(* CODESYS project CtaAppStufenManagement_4.0.0.1.library
   Description: Stufenmanagement Library der CTA
   Version: 4.0.0.1
   Title: CtaAppStufenManagement
   Author: SIS
   DocFormat: reStructuredText
   LanguageModelAttribute: qualified-access-only
   Placeholder: CtaAppStufenManagement
   DefaultNamespace: CtaAppStufenManagement
   CompiledLibraryCompatibilityVersion: CODESYS V3.5 SP16 Patch 3
   Company: CTA

Project tree, tasks and I/O mapping:
  libraries: Standard, 3.5.18.0 (System); CtaAppBasic, 1.0.0.1 (CTA); CtaAppBmk, 2.0.0.0 (CTA); CtaSysConfig, 2.0.0.0 (CTA); VisuDialogs, 3.5.16.20 (System); VisuSymbols, 4.5.0.0 (System); CtaVisHelp, 2.0.0.0 (CTA); CtaVisSymbols, 2.0.0.1 (CTA); CtaSysTypes, 1.0.0.0 (CTA)
  40 Visualizations/
    visualisation VIS_Manager_rEck
    Dialog/
      visualisation DIA_MANAGERCONFIG
    visualisation VIS_Manager
  00000000-0000-0000-0000-000000000000|D:\CoDeSys\LibrariesV3\trunk\Intern\CAA\CAA Template\3.4.0.0 draft\Placeholder.xml
  00000000-0000-0000-0000-000000000000|D:\CoDeSys\LibrariesV3\trunk\Intern\CAA\CAA Template\3.2.0.3 draft\Prefix.pdf
  00000000-0000-0000-0000-000000000000|D:\CoDeSys\LibrariesV3\trunk\Intern\CAA\CAA Template\3.5.2.0 draft\Placeholder.xml
  20 Structs/
    data type TYPE_OF_ENGINE_MANAGEMENT
    data type scParameter
  50 Images/
  10 Documenation/
    global variables VersionHistory
    global variables readMe
  21 Interface/
    Group/
      GroupBase/
        interface ITF_GROUPBASE: IS_NOT_RELEVANT_TO_CHECK, set_acknowledge_substate, acknowledge_substate, acknowledge, set_acknowledge, acknowledge_old, acknowledge_substate_old, IS_NOT_RELEVANT_TO_RELEASE, IS_ADDED_TO_NESSESARY, check, set_check, set_check_substate, check_substate, check_old, check_substate_old, release, set_release, set_release_next, set_release_substate, release_substate, release_old, release_substate_old, release_next, release_next_old, IS_NOT_RELEVANT_TO_ACKNOWLEDGE, available_substate, set_available_substate, set_available, available, available_old, available_substate_old, set_demand, demand, demand_old
      GroupLeader/
        Circuit/
          interface ITF_CIRCUIT: GET_ANZ_AVAIABLE, GET_ANZ_ACKNOWLEDGE, GET_ANZ_RELEASE, CIRCUIT_NR, ALL_OFF, IS_RELEVANT_TO_RELEASE, GET_ENGINE_STATE, RELEASE_ENGINE, LOWERBOUND, UPPERBOUND, GET_ANZ_LOCKDOWN, SET_HZ_SCALE, SET_ENGINE_STATE, prorRelease, GET_SUM_ACKNOWLEDGE_HZ
      GroupMember/
        Hydraulics/
          interface ITF_HYDRA: MEMBER_OF
    Manager/
      interface ITF_MANAGER: ADD_CLIENT
  11 Library Parameter/
  12 Konstanten/
    global variables GVL_CONSTANT
  60 Textlisten/
    text list TypeOfEngineManagement
  13 Globale Variablen/
  text list GlobalTextList
  5ce3da45-db07-42e7-a21c-a00fff4ed8f6|C:\Users\sis\Downloads\dip-switch.svg
  5ce3da45-db07-42e7-a21c-a00fff4ed8f6|C:\Users\sis\Downloads\lightning-bolt-circle.svg
  30 Program Organization Units/
    Group/
      GroupBase/
        function block GROUPBASE [ST]: IS_NOT_RELEVANT_TO_CHECK, IS_NOT_RELEVANT_TO_RELEASE, set_acknowledge, set_acknowledge_substate, acknowledge, acknowledge_substate, acknowledge_old, acknowledge_substate_old, available_substate, available, set_available, set_available_substate, available_old, available_substate_old, check_substate, set_check_substate, check, set_check, check_old, check_substate_old, set_release_next, release, release_substate, set_release, set_release_substate, release_next, release_next_old, release_old, release_substate_old, IS_NOT_RELEVANT_TO_ACKNOWLEDGE, set_demand, demand, demand_old, IS_ADDED_TO_NESSESARY
      GroupLeader/
        Help/
          function block ENGINE [ST]: GET_ANZ_AVAIABLE, GET_ANZ_ACKNOWLEDGE, GET_ANZ_RELEASE, GET_ANZ_LOCKDOWN, SET_ENGINE_STATE, GET_ENGINE_STATE, RELEASE_ENGINE, LOWERBOUND, UPPERBOUND, SET_HZ_SCALE, GET_ANZ_ENABLED, GET_SUM_ACKNOWLEDGE_HZ
        Circuit/
          function block CIRCUIT [ST]: IS_RELEVANT_TO_RELEASE, SET_ENGINE_STATE, GET_ANZ_AVAIABLE, GET_ANZ_ACKNOWLEDGE, GET_ANZ_RELEASE, CIRCUIT_NR, ALL_OFF, GET_ENGINE_STATE, RELEASE_ENGINE, LOWERBOUND, UPPERBOUND, GET_ANZ_LOCKDOWN, SET_HZ_SCALE, prorRelease, GET_ANZ_ENABLED, GET_SUM_ACKNOWLEDGE_HZ
      GroupMember/
        Help/
          function block GROUPMEMBER [ST]
        Hydraulics/
          function block HYDRA [ST]: MEMBER_OF, FB_INIT
    Manager/
      function block MANAGER [ST]: CHECK, set_check_of_group, set_check_substate_of_group, get_next_engine_to_start, get_next_engine_to_stopp, engine_management_start_run_1_by_1, engine_management_start_run_equal, engine_management_stopp_run_1_by_1, engine_management_stopp_run_equal, ENGINE_MANAGEMENT, UPDATE_AT_THE_END, ACKNOWLEDGE, check_acknowledge_of_group, check_acknowledge_substate_of_group, RELEASE, set_release_of_group, set_release_substate_of_group, set_release_next_of_group, LOCKDOWN, AVAIABLE, check_available_of_group, check_available_substate_of_group, ADD_CLIENT, actParameter, FB_INIT, DEMAND, set_priority_array, init_priority_array_with_ignore_state
  5ce3da45-db07-42e7-a21c-a00fff4ed8f6|C:\Users\sis\Downloads\sine-wave.svg
  5ce3da45-db07-42e7-a21c-a00fff4ed8f6|C:\Users\sis\Downloads\eye.svg
  5ce3da45-db07-42e7-a21c-a00fff4ed8f6|C:\Users\sis\Downloads\lan.svg
*)

// 20 Structs/TYPE_OF_ENGINE_MANAGEMENT
{attribute 'qualified_only'}
TYPE TYPE_OF_ENGINE_MANAGEMENT :
(
	RUN_1BY1 	:= 0,
	RUN_EQUAL	:= 1
);
END_TYPE

// 20 Structs/scParameter
TYPE scParameter :
	STRUCT
		fbtZuschaltSperrzeit		:	CtaSysConfig.fbTIME;
		fbiTypeOfEngineManagement	:	CtaSysConfig.fbINT;
	END_STRUCT
END_TYPE

// 10 Documenation/VersionHistory
(* 

.. image:: ../../Images/CTA_Logo.jpg
   :align: right
   :width: 15% 

**Vorlage**   


============ =========== =========== ============================================
**Date**     **Version** **Author**  **Change**
------------ ----------- ----------- --------------------------------------------
04.03.2021   0.0.0.0     SIS         Vorlage erstellt

============ =========== =========== ============================================


*)
VAR_GLOBAL
    stInfo : STRING:= '0.0.0.0, Vorlage, CTA';
END_VAR

// 10 Documenation/readMe
(*

**ReadMe**
 
|	**Empfehlung**
|
|	Die Bibliothek CtaAppStufenManagement dient dem Management der ganzen Maschine, sie Schaltet beispielsweise Kreise und Stufen frei.
|	Instanzieren Sie den CtaAppStufenManagement.MANAGER in ihrem Funktionsbaustein oder POU beispielsweise als Manager
|	Deklarieren Sie die Struktur Variable welche als Parameter und zur ansteuerung dienen wie im Code beispiel.
|  
| *Beispiel* 

+-----------------------+---------------------------------------------------------------------------------------------------------------------------------------------------------------------------------------------------------------------------------------------------------------------------------------------------------------------------------------------------------------------------------------------------------------------------------------+
| Beschreibung          |  Code                                                                                                                                                                                                                                                                                                                                                                                                                                 |
+=======================+=======================================================================================================================================================================================================================================================================================================================================================================================================================================+
| Pou oder SmFb         | .. code-block:: codesys                                                                                                                                                                                                                                                                                                                                                                                                               |
|                       |                                                                                                                                                                                                                                                                                                                                                                                                                                       |
|                       |	// Deklaration als VAR im POU oder dem selbsterstellten Funktionsbaustein                                                                                                                                                                                                                                                                                                                                                       	|
|                       |   VAR   																																																																																																								|
|						|	    (*Maschinen Management*)																																																		 																																																|
|						|		MANAGER			: CtaAppStufenManagement.MANAGER;                                                                                                                                                                                                                                                                                                                                                             				 	|
|						|																																																																																																										|
+-----------------------+---------------------------------------------------------------------------------------------------------------------------------------------------------------------------------------------------------------------------------------------------------------------------------------------------------------------------------------------------------------------------------------------------------------------------------------+
| Code für Init         | .. code-block:: codesys                                                                                                                                                                                                                                                                                                                                                                                                               |
|                       |   																																																																																																									|
| 						|	// Kopieren des nachfolgenden Codes in eine Action zur Initialisierung der Parameter. Zum Beispiel actConfig.																																																																														|
|                       |	{region "Maschinen Management"}                                                                                                                                                                                                                                                                                                                                                                                                     |
|						|		MANAGER.scParameter.fbtZuschaltSperrzeit               		(_wertInit :=	 T#5m														);		//P1 Zeit die vergeht bis die nächste Stufe zugeschalten werden kann																																																			|
|						|		MANAGER.scParameter.fbiTypeOfEngineManagement				(_wertInit :=	 	0		, _minInit :=			, _maxInit :=			);		//P2 0 = Ausschöpfung des Kreises / 1 = Beliebig nach verfügbarkeit																																																				| 
|						|	{endregion}                                                                                                                                                      																																																																	| 
+-----------------------+---------------------------------------------------------------------------------------------------------------------------------------------------------------------------------------------------------------------------------------------------------------------------------------------------------------------------------------------------------------------------------------------------------------------------------------+
*)                                                                                                                                                                                                                                                                                                                                                                                                                                                               
 VAR_GLOBAL                                                                                                                                                                                                                                                                                                                                                                                                                                                      
    xReadMeDone              :   BOOL;                                                                                                                                                                                                                                                                                                                                                                                                                           
END_VAR

// 12 Konstanten/GVL_CONSTANT
{attribute 'qualified_only'}
VAR_GLOBAL CONSTANT
	MAX_GROUPS	:	USINT	:= 4;
	MAX_ENGINE	:	USINT	:= 4;
END_VAR

// 21 Interface/Group/GroupBase/ITF_GROUPBASE
INTERFACE ITF_GROUPBASE EXTENDS __SYSTEM.IQueryInterface

{attribute 'monitoring':='call'}
PROPERTY IS_NOT_RELEVANT_TO_CHECK : BOOL
GET
END_GET
SET
END_SET
END_PROPERTY

METHOD set_acknowledge_substate
VAR_INPUT
	_en_acknowledge_substate		:	INT;
END_VAR
END_METHOD

{attribute 'monitoring':='call'}
PROPERTY acknowledge_substate : INT
GET
END_GET
END_PROPERTY

{attribute 'monitoring':='call'}
PROPERTY acknowledge : INT
GET
END_GET
END_PROPERTY

METHOD set_acknowledge
VAR_INPUT
	_en_acknowledge		:	INT;
END_VAR
END_METHOD

{attribute 'monitoring':='call'}
PROPERTY acknowledge_old : INT
GET
END_GET
END_PROPERTY

{attribute 'monitoring':='call'}
PROPERTY acknowledge_substate_old : INT
GET
END_GET
END_PROPERTY

{attribute 'monitoring':='call'}
PROPERTY IS_NOT_RELEVANT_TO_RELEASE : BOOL
GET
END_GET
SET
END_SET
END_PROPERTY

PROPERTY IS_ADDED_TO_NESSESARY : BOOL
SET
END_SET
GET
END_GET
END_PROPERTY

{attribute 'monitoring':='call'}
PROPERTY check : INT
GET
END_GET
END_PROPERTY

METHOD set_check
VAR_INPUT
	_en_check			:	INT;
END_VAR
END_METHOD

METHOD set_check_substate
VAR_INPUT
	_en_check_substate				:	INT;
END_VAR
END_METHOD

{attribute 'monitoring':='call'}
PROPERTY check_substate : INT
GET
END_GET
END_PROPERTY

{attribute 'monitoring':='call'}
PROPERTY check_old : INT
GET
END_GET
END_PROPERTY

{attribute 'monitoring':='call'}
PROPERTY check_substate_old : INT
GET
END_GET
END_PROPERTY

{attribute 'monitoring':='call'}
PROPERTY release : INT
GET
END_GET
END_PROPERTY

METHOD set_release
VAR_INPUT
	_en_release			:	INT;
END_VAR
END_METHOD

METHOD set_release_next
VAR_INPUT
	_en_release_next	:	INT;
END_VAR
END_METHOD

METHOD set_release_substate
VAR_INPUT
	_en_release_substate	:	INT;
END_VAR
END_METHOD

{attribute 'monitoring':='call'}
PROPERTY release_substate : INT
GET
END_GET
END_PROPERTY

{attribute 'monitoring':='call'}
PROPERTY release_old : INT
GET
END_GET
END_PROPERTY

{attribute 'monitoring':='call'}
PROPERTY release_substate_old : INT
GET
END_GET
END_PROPERTY

PROPERTY release_next : INT
GET
END_GET
END_PROPERTY

PROPERTY release_next_old : INT
GET
END_GET
END_PROPERTY

{attribute 'monitoring':='call'}
PROPERTY IS_NOT_RELEVANT_TO_ACKNOWLEDGE : BOOL
SET
END_SET
GET
END_GET
END_PROPERTY

{attribute 'monitoring':='call'}
PROPERTY available_substate : INT
GET
END_GET
END_PROPERTY

METHOD set_available_substate
VAR_INPUT
	_en_avaiable_substate	:	INT;
END_VAR
END_METHOD

METHOD set_available
VAR_INPUT
	_en_avaiable		:	INT;
END_VAR
END_METHOD

{attribute 'monitoring':='call'}
PROPERTY available : INT
GET
END_GET
END_PROPERTY

{attribute 'monitoring':='call'}
PROPERTY available_old : INT
GET
END_GET
END_PROPERTY

{attribute 'monitoring':='call'}
PROPERTY available_substate_old : INT
GET
END_GET
END_PROPERTY

METHOD set_demand
VAR_INPUT
	_en_demand			:	INT;
END_VAR
END_METHOD

{attribute 'monitoring':='call'}
PROPERTY demand : INT
GET
END_GET
END_PROPERTY

{attribute 'monitoring':='call'}
PROPERTY demand_old : INT
GET
END_GET
END_PROPERTY

END_INTERFACE

// 21 Interface/Manager/ITF_MANAGER
INTERFACE ITF_MANAGER EXTENDS __SYSTEM.IQueryInterface

METHOD ADD_CLIENT : BOOL
VAR_INPUT
	ITF_GROUP_BASE_IN	:	ITF_GROUPBASE;
END_VAR
END_METHOD

END_INTERFACE

// 21 Interface/Group/GroupLeader/Circuit/ITF_CIRCUIT
INTERFACE ITF_CIRCUIT EXTENDS ITF_GROUPBASE

PROPERTY GET_ANZ_AVAIABLE : UINT
GET
END_GET
END_PROPERTY

PROPERTY GET_ANZ_ACKNOWLEDGE : UINT
GET
END_GET
END_PROPERTY

PROPERTY GET_ANZ_RELEASE : UINT
GET
END_GET
END_PROPERTY

PROPERTY CIRCUIT_NR : USINT
GET
END_GET
END_PROPERTY

METHOD ALL_OFF : BOOL
VAR_INPUT
END_VAR
END_METHOD

PROPERTY IS_RELEVANT_TO_RELEASE : BOOL
GET
END_GET
SET
END_SET
END_PROPERTY

METHOD GET_ENGINE_STATE : BOOL
VAR_INPUT
	usiNr				:	USINT;
END_VAR
VAR_OUTPUT	    	
	xAvaiable			:	BOOL;
	xRelease			:	BOOL;
	rRelease			:	REAL;
	xAcknowledge		:	BOOL;
	rAcknowledgeHz		:	REAL;
	xLockDown			:	BOOL;
	udiRunTime			:	UDINT;
	udiRunTimeTillOn	:	UDINT;
END_VAR
END_METHOD

METHOD RELEASE_ENGINE
VAR_INPUT
	usiNr		:	USINT;
	xRelease	:	BOOL;
END_VAR
END_METHOD

PROPERTY LOWERBOUND : DINT
GET
END_GET
END_PROPERTY

PROPERTY UPPERBOUND : DINT
GET
END_GET
END_PROPERTY

PROPERTY GET_ANZ_LOCKDOWN : UINT
GET
END_GET
END_PROPERTY

METHOD SET_HZ_SCALE
VAR_INPUT
	scHz		:	CtaSysTypes.scHzParameter;
END_VAR
END_METHOD

METHOD SET_ENGINE_STATE 
VAR_INPUT
	usiNr		:	USINT;
	xEnabled	:	BOOL;
	xAvaiable	:	BOOL;
	xAcknowledge:	BOOL;
	rAcknowledgeHz:	REAL;
	xLockDown	:	BOOL;
	rNewRelease	:	REAL;
END_VAR
VAR_OUTPUT
	xRelease	:	BOOL;
	rRelease	:	REAL;
	scHz		:	CtaSysTypes.scHzParameter;
END_VAR
END_METHOD

PROPERTY prorRelease : REAL
SET
END_SET
GET
END_GET
END_PROPERTY

PROPERTY GET_SUM_ACKNOWLEDGE_HZ : REAL
GET
END_GET
END_PROPERTY

END_INTERFACE

// 21 Interface/Group/GroupMember/Hydraulics/ITF_HYDRA
INTERFACE ITF_HYDRA EXTENDS ITF_GROUPBASE

METHOD MEMBER_OF : BOOL
VAR_INPUT
	usiGROUP_NR	:	USINT;
END_VAR
END_METHOD

END_INTERFACE

// 30 Program Organization Units/Group/GroupBase/GROUPBASE
FUNCTION_BLOCK GROUPBASE IMPLEMENTS ITF_GROUPBASE
VAR_INPUT
	ITF_MANAGER_IN			:	ITF_MANAGER;
END_VAR           		         		
VAR                 		
	en_check						:	INT;
	en_check_substate				:	INT;
	en_check_old					:	INT;
	en_check_substate_old			:	INT;	
	en_release						:	INT;
	en_release_substate				:	INT;
	en_release_next					: 	INT;	
	en_release_old					:	INT;
	en_release_substate_old			:	INT;
	en_release_next_old				: 	INT;
	en_acknowledge					:	INT;
	en_acknowledge_substate			:	INT;    
	en_acknowledge_old				:	INT;
	en_acknowledge_substate_old		:	INT;   				
	en_available					:	INT;
	en_available_substate			:	INT;
	en_available_old				:	INT;
	en_available_substate_old		:	INT;
	en_demand						:	INT;
	en_demand_old					:	INT;
	_Is_Not_Relevant_To_Release		:	BOOL;
	_Is_Not_Relevant_To_Check		:	BOOL;
	_Is_Not_Relevant_To_Acknowledge :	BOOL;
	ITF_MANAGER_OLD					:	ITF_MANAGER;
	xIsAddedToNessesary				:	BOOL;
END_VAR

IF __QUERYINTERFACE(ITF_MANAGER_IN,ITF_MANAGER_IN) THEN
	IF ITF_MANAGER_IN <> ITF_MANAGER_OLD OR NOT xIsAddedToNessesary THEN
		xIsAddedToNessesary := FALSE;
		ITF_MANAGER_IN.ADD_CLIENT(THIS^);	
		ITF_MANAGER_OLD := ITF_MANAGER_IN;
	END_IF;
END_IF;

{attribute 'monitoring':='call'}
PROPERTY IS_NOT_RELEVANT_TO_CHECK : BOOL
GET
IS_NOT_RELEVANT_TO_CHECK := _Is_Not_Relevant_To_Check;
END_GET
SET
_Is_Not_Relevant_To_Check := IS_NOT_RELEVANT_TO_CHECK;
END_SET
END_PROPERTY

{attribute 'monitoring':='call'}
PROPERTY IS_NOT_RELEVANT_TO_RELEASE : BOOL
GET
IS_NOT_RELEVANT_TO_RELEASE := _Is_Not_Relevant_To_Release;
END_GET
SET
_Is_Not_Relevant_To_Release := IS_NOT_RELEVANT_TO_RELEASE;
END_SET
END_PROPERTY

METHOD set_acknowledge
VAR_INPUT
	_en_acknowledge		:	INT;
END_VAR
IF _en_acknowledge <> en_acknowledge THEN
	en_acknowledge_old := en_acknowledge;
	en_acknowledge := _en_acknowledge;
END_IF;
END_METHOD

METHOD set_acknowledge_substate
VAR_INPUT
	_en_acknowledge_substate		:	INT;
END_VAR
IF _en_acknowledge_substate <> en_acknowledge_substate THEN
	en_acknowledge_substate_old := _en_acknowledge_substate;
	en_acknowledge_substate := _en_acknowledge_substate;
END_IF;
END_METHOD

{attribute 'monitoring':='call'}
PROPERTY acknowledge : INT
GET
acknowledge := en_acknowledge;
END_GET
END_PROPERTY

{attribute 'monitoring':='call'}
PROPERTY acknowledge_substate : INT
GET
acknowledge_substate := en_acknowledge_substate;
END_GET
END_PROPERTY

{attribute 'monitoring':='call'}
PROPERTY acknowledge_old : INT
GET
acknowledge_old := en_acknowledge_old;
END_GET
END_PROPERTY

{attribute 'monitoring':='call'}
PROPERTY acknowledge_substate_old : INT
GET
acknowledge_substate_old := en_acknowledge_substate_old;
END_GET
END_PROPERTY

{attribute 'monitoring':='call'}
PROPERTY available_substate : INT
GET
available_substate := en_available_substate;
END_GET
END_PROPERTY

{attribute 'monitoring':='call'}
PROPERTY available : INT
GET
available := en_available;
END_GET
END_PROPERTY

METHOD set_available
VAR_INPUT
	_en_avaiable		:	INT;
END_VAR
IF _en_avaiable <> en_available THEN
	en_available_old := en_available;
	en_available := _en_avaiable;
END_IF;
END_METHOD

METHOD set_available_substate
VAR_INPUT
	_en_avaiable_substate	:	INT;
END_VAR
IF _en_avaiable_substate <> en_available_substate THEN
	en_available_substate_old := en_available_substate;
	en_available_substate := _en_avaiable_substate;
END_IF;
END_METHOD

{attribute 'monitoring':='call'}
PROPERTY available_old : INT
GET
available_old := en_available_old;
END_GET
END_PROPERTY

{attribute 'monitoring':='call'}
PROPERTY available_substate_old : INT
GET
available_substate_old := en_available_substate_old;
END_GET
END_PROPERTY

{attribute 'monitoring':='call'}
PROPERTY check_substate : INT
GET
check_substate := en_check_substate;
END_GET
END_PROPERTY

METHOD set_check_substate
VAR_INPUT
	_en_check_substate				:	INT;
END_VAR
IF _en_check_substate <> en_check_substate THEN
	en_check_substate_old := en_check_substate;
	en_check_substate := _en_check_substate;
END_IF;
END_METHOD

{attribute 'monitoring':='call'}
PROPERTY check : INT
GET
check := en_check;
END_GET
END_PROPERTY

METHOD set_check
VAR_INPUT
	_en_check			:	INT;
END_VAR
IF _en_check <> en_check THEN
	en_check_old := en_check;
	en_check := _en_check;
END_IF;
END_METHOD

{attribute 'monitoring':='call'}
PROPERTY check_old : INT
GET
check_old := en_check_old;
END_GET
END_PROPERTY

{attribute 'monitoring':='call'}
PROPERTY check_substate_old : INT
GET
check_substate_old := en_check_substate_old;
END_GET
END_PROPERTY

METHOD set_release_next
VAR_INPUT
	_en_release_next	:	INT;
END_VAR
IF _en_release_next <> en_release_next THEN
	en_release_next_old := en_release_next;
	en_release_next := _en_release_next;
END_IF;
END_METHOD

{attribute 'monitoring':='call'}
PROPERTY release : INT
GET
release := en_release;
END_GET
END_PROPERTY

{attribute 'monitoring':='call'}
PROPERTY release_substate : INT
GET
release_substate := en_release_substate;
END_GET
END_PROPERTY

METHOD set_release
VAR_INPUT
	_en_release			:	INT;
END_VAR
IF _en_release <> en_release THEN
	en_release_old := en_release;
	en_release := _en_release;
END_IF
END_METHOD

METHOD set_release_substate
VAR_INPUT
	_en_release_substate	:	INT;
END_VAR
IF _en_release_substate <> en_release_substate THEN
	en_release_substate_old := en_release_substate;
	en_release_substate := _en_release_substate;
END_IF;
END_METHOD

PROPERTY release_next : INT
GET
release_next := en_release_next;
END_GET
END_PROPERTY

PROPERTY release_next_old : INT
GET
release_next_old := en_release_next_old;
END_GET
END_PROPERTY

{attribute 'monitoring':='call'}
PROPERTY release_old : INT
GET
release_old := en_release_old;
END_GET
END_PROPERTY

{attribute 'monitoring':='call'}
PROPERTY release_substate_old : INT
GET
release_substate_old := en_release_substate_old;
END_GET
END_PROPERTY

{attribute 'monitoring':='call'}
PROPERTY IS_NOT_RELEVANT_TO_ACKNOWLEDGE : BOOL
GET
IS_NOT_RELEVANT_TO_ACKNOWLEDGE := _Is_Not_Relevant_To_Acknowledge;
END_GET
SET
_Is_Not_Relevant_To_Acknowledge := IS_NOT_RELEVANT_TO_ACKNOWLEDGE;
END_SET
END_PROPERTY

METHOD set_demand
VAR_INPUT
	_en_demand			:	INT;
END_VAR
IF _en_demand <> en_demand THEN
	en_demand_old := en_demand;
	en_demand := _en_demand;
END_IF;
END_METHOD

{attribute 'monitoring':='call'}
PROPERTY demand : INT
GET
demand := en_demand;
END_GET
END_PROPERTY

{attribute 'monitoring':='call'}
PROPERTY demand_old : INT
GET
demand_old := en_demand_old;
END_GET
END_PROPERTY

PROPERTY IS_ADDED_TO_NESSESARY : BOOL
GET
IS_ADDED_TO_NESSESARY := xIsAddedToNessesary;
END_GET
SET
xIsAddedToNessesary := IS_ADDED_TO_NESSESARY;
END_SET
END_PROPERTY

END_FUNCTION_BLOCK

// 30 Program Organization Units/Group/GroupLeader/Circuit/CIRCUIT
FUNCTION_BLOCK CIRCUIT EXTENDS GROUPBASE IMPLEMENTS ITF_CIRCUIT
VAR_INPUT
	usiNr	:	USINT;
END_VAR
VAR_OUTPUT
END_VAR
VAR
	xRelease					:	BOOL;
	rRelease					:	REAL;
	xIsRelevantToRelease		:	BOOL;
	ENGINE						:	ENGINE;
	diFor						:	DINT;
END_VAR

SUPER^();

PROPERTY IS_RELEVANT_TO_RELEASE : BOOL
SET
xIsRelevantToRelease := IS_RELEVANT_TO_RELEASE;
END_SET
GET
IS_RELEVANT_TO_RELEASE := xIsRelevantToRelease;
END_GET
END_PROPERTY

METHOD SET_ENGINE_STATE 
VAR_INPUT
	usiNr		:	USINT;
	xEnabled	:	BOOL;
	xAvaiable	:	BOOL;
	xAcknowledge:	BOOL;
	rAcknowledgeHz:	REAL;
	xLockDown	:	BOOL;
	rNewRelease	:	REAL;
END_VAR
VAR_OUTPUT
	xRelease	:	BOOL;
	rRelease	:	REAL;
	scHz		:	CtaSysTypes.scHzParameter;
END_VAR
ENGINE.SET_ENGINE_STATE(usiNr 			:= usiNr,
						xEnabled		:= xEnabled,
						xAvaiable 		:= xAvaiable,
						xAcknowledge	:= xAcknowledge,
						rAcknowledgeHz	:= rAcknowledgeHz,
						xLockDown		:= xLockDown,
						rNewRelease		:= rNewRelease,
						xRelease		=> xRelease,
						rRelease		=> rRelease,
						scHz			=> scHz);
END_METHOD

PROPERTY GET_ANZ_AVAIABLE : UINT
GET
VAR
	diForTemp	:	DINT;
END_VAR
GET_ANZ_AVAIABLE := ENGINE.GET_ANZ_AVAIABLE;
END_GET
END_PROPERTY

PROPERTY GET_ANZ_ACKNOWLEDGE : UINT
GET
VAR
	diForTemp	:	DINT;
END_VAR
GET_ANZ_ACKNOWLEDGE := ENGINE.GET_ANZ_ACKNOWLEDGE;
END_GET
END_PROPERTY

PROPERTY GET_ANZ_RELEASE : UINT
GET
VAR
	diForTemp	:	DINT;
END_VAR
GET_ANZ_RELEASE := ENGINE.GET_ANZ_RELEASE;
END_GET
END_PROPERTY

PROPERTY CIRCUIT_NR : USINT
GET
CIRCUIT_NR := usiNr;
END_GET
END_PROPERTY

METHOD ALL_OFF : BOOL
VAR_INPUT
END_VAR
VAR
	diLowerBound	:	DINT;
	diUpperBound	:	DINT;
	diForTemp1		:	DINT;
END_VAR
(* Stopp ALL *)
FOR diForTemp1 := ENGINE.LOWERBOUND TO ENGINE.UPPERBOUND DO
	ENGINE.RELEASE_ENGINE(TO_USINT(diForTemp1),FALSE);
END_FOR;
END_METHOD

METHOD GET_ENGINE_STATE : BOOL
VAR_INPUT
	usiNr		:	USINT;
END_VAR
VAR_OUTPUT	    	
	xAvaiable			:	BOOL;
	xRelease			:	BOOL;
	rRelease			:	REAL;
	xAcknowledge		:	BOOL;
	rAcknowledgeHz		:	REAL;
	xLockDown			:	BOOL;
	udiRunTime			:	UDINT;
	udiRunTimeTillOn	:	UDINT;
END_VAR
ENGINE.GET_ENGINE_STATE(usiNr 				:= usiNr,
						xAvaiable			=> xAvaiable,
						xRelease			=> xRelease,
						rRelease			=> rRelease,
						xAcknowledge		=> xAcknowledge,
						rAcknowledgeHz		=> rAcknowledgeHz,
						xLockDown			=> xLockDown,
						udiRunTime			=> udiRunTime,
						udiRunTimeTillOn	=> udiRunTimeTillOn);
END_METHOD

METHOD RELEASE_ENGINE
VAR_INPUT
	usiNr		:	USINT;
	xRelease	:	BOOL;
END_VAR
ENGINE.RELEASE_ENGINE(	usiNr		:= usiNr,
						xRelease 	:= xRelease);
END_METHOD

PROPERTY LOWERBOUND : DINT
GET
LOWERBOUND := ENGINE.LOWERBOUND;
END_GET
END_PROPERTY

PROPERTY UPPERBOUND : DINT
GET
UPPERBOUND := ENGINE.UPPERBOUND;
END_GET
END_PROPERTY

PROPERTY GET_ANZ_LOCKDOWN : UINT
GET
GET_ANZ_LOCKDOWN := ENGINE.GET_ANZ_LOCKDOWN;
END_GET
END_PROPERTY

METHOD SET_HZ_SCALE
VAR_INPUT
	scHz		:	CtaSysTypes.scHzParameter;
END_VAR
ENGINE.SET_HZ_SCALE(scHz);
END_METHOD

PROPERTY prorRelease : REAL
GET
prorRelease := rRelease;
END_GET
SET
rRelease := prorRelease;
END_SET
END_PROPERTY

PROPERTY GET_ANZ_ENABLED : UINT
GET
VAR
	diForTemp	:	DINT;
END_VAR
GET_ANZ_ENABLED := ENGINE.GET_ANZ_ENABLED;
END_GET
END_PROPERTY

PROPERTY GET_SUM_ACKNOWLEDGE_HZ : REAL
GET
VAR
	diForTemp	:	DINT;
END_VAR
GET_SUM_ACKNOWLEDGE_HZ := ENGINE.GET_SUM_ACKNOWLEDGE_HZ;
END_GET
END_PROPERTY

END_FUNCTION_BLOCK

// 30 Program Organization Units/Group/GroupLeader/Help/ENGINE
FUNCTION_BLOCK ENGINE
VAR_INPUT
END_VAR
VAR_OUTPUT
END_VAR
VAR
	scHzAll				:	CtaSysTypes.scHzParameter;
	AY_XENABLED			:	ARRAY[1..GVL_CONSTANT.MAX_ENGINE] OF BOOL;
	AY_XRELEASE			:	ARRAY[1..GVL_CONSTANT.MAX_ENGINE] OF BOOL;
	AY_RRELEASE			:	ARRAY[1..GVL_CONSTANT.MAX_ENGINE] OF REAL;
	AY_XAVAIABLE		:	ARRAY[1..GVL_CONSTANT.MAX_ENGINE] OF BOOL;
	AY_XACKNOWLEDGE		:	ARRAY[1..GVL_CONSTANT.MAX_ENGINE] OF BOOL;
	AY_XACKNOWLEDGEOLD	:	ARRAY[1..GVL_CONSTANT.MAX_ENGINE] OF BOOL;
	AY_RACKNOWLEDGE		:	ARRAY[1..GVL_CONSTANT.MAX_ENGINE] OF REAL;
	AY_LOCKDOWN			:	ARRAY[1..GVL_CONSTANT.MAX_ENGINE] OF BOOL;
	AY_RUN_TIME			:	ARRAY[1..GVL_CONSTANT.MAX_ENGINE] OF UDINT;
	AY_RUN_TIME_TILL_ON	:	ARRAY[1..GVL_CONSTANT.MAX_ENGINE] OF UDINT;
	AY_TON_RUN_TIME		:	ARRAY[1..GVL_CONSTANT.MAX_ENGINE] OF Standard.TON;
END_VAR

PROPERTY GET_ANZ_AVAIABLE : UINT
GET
VAR
	diForTemp	:	DINT;
END_VAR
GET_ANZ_AVAIABLE := 0;
FOR diForTemp := LOWER_BOUND(AY_XAVAIABLE,1) TO UPPER_BOUND(AY_XAVAIABLE,1) DO
	IF AY_XAVAIABLE[diForTemp] THEN
		GET_ANZ_AVAIABLE := GET_ANZ_AVAIABLE + 1;
	END_IF;
END_FOR;
END_GET
END_PROPERTY

PROPERTY GET_ANZ_ACKNOWLEDGE : UINT
GET
VAR
	diForTemp	:	DINT;
END_VAR
GET_ANZ_ACKNOWLEDGE := 0;
FOR diForTemp := LOWER_BOUND(AY_XACKNOWLEDGE,1) TO UPPER_BOUND(AY_XACKNOWLEDGE,1) DO
	IF AY_XACKNOWLEDGE[diForTemp] THEN
		GET_ANZ_ACKNOWLEDGE := GET_ANZ_ACKNOWLEDGE + 1;
	END_IF;
END_FOR;
END_GET
END_PROPERTY

PROPERTY GET_ANZ_RELEASE : UINT
GET
VAR
	diForTemp	:	DINT;
END_VAR
GET_ANZ_RELEASE := 0;
FOR diForTemp := LOWER_BOUND(AY_XRELEASE,1) TO UPPER_BOUND(AY_XRELEASE,1) DO
	IF AY_XRELEASE[diForTemp] THEN
		GET_ANZ_RELEASE := GET_ANZ_RELEASE + 1;
	END_IF;
END_FOR;
END_GET
END_PROPERTY

PROPERTY GET_ANZ_LOCKDOWN : UINT
GET
VAR
	diForTemp	:	DINT;
END_VAR
GET_ANZ_LOCKDOWN := 0;
FOR diForTemp := LOWER_BOUND(AY_LOCKDOWN,1) TO UPPER_BOUND(AY_LOCKDOWN,1) DO
	IF AY_LOCKDOWN[diForTemp] THEN
		GET_ANZ_LOCKDOWN := GET_ANZ_LOCKDOWN + 1;
	END_IF;
END_FOR;
END_GET
END_PROPERTY

METHOD SET_ENGINE_STATE 
VAR_INPUT
	usiNr			:	USINT;
	xEnabled		:	BOOL;
	xAvaiable		:	BOOL;
	xAcknowledge	:	BOOL;
	rAcknowledgeHz	:	REAL;
	xLockDown		:	BOOL;
	rNewRelease		:	REAL;
END_VAR
VAR_OUTPUT
	xRelease	:	BOOL;
	rRelease	:	REAL;
	scHz		:	CtaSysTypes.scHzParameter;
END_VAR
(* Enabled *)
IF usiNr >= LOWER_BOUND(AY_XENABLED,1) AND usiNr <= UPPER_BOUND(AY_XENABLED,1) THEN
	AY_XENABLED[usiNr] := xEnabled;
END_IF;

(* Avaiable *)
IF usiNr >= LOWER_BOUND(AY_XAVAIABLE,1) AND usiNr <= UPPER_BOUND(AY_XAVAIABLE,1) THEN
	AY_XAVAIABLE[usiNr] := xAvaiable;
END_IF;

(* Acknowledge *)
IF usiNr >= LOWER_BOUND(AY_XACKNOWLEDGE,1) AND usiNr <= UPPER_BOUND(AY_XACKNOWLEDGE,1) THEN
	AY_XACKNOWLEDGEOLD[usiNr] 	:= AY_XACKNOWLEDGE[usiNr];
	AY_XACKNOWLEDGE[usiNr] 		:= xAcknowledge;
END_IF;
IF usiNr >= LOWER_BOUND(AY_RACKNOWLEDGE,1) AND usiNr <= UPPER_BOUND(AY_RACKNOWLEDGE,1) THEN
	AY_RACKNOWLEDGE[usiNr] := rAcknowledgeHz;
END_IF

(* LockDown *)
IF usiNr >= LOWER_BOUND(AY_LOCKDOWN,1) AND usiNr <= UPPER_BOUND(AY_LOCKDOWN,1) THEN
	AY_LOCKDOWN[usiNr] := xLockDown;
	IF xLockDown THEN
		AY_XRELEASE[usiNr] := FALSE;
	END_IF;
END_IF;

(* Release *)
IF usiNr >= LOWER_BOUND(AY_XRELEASE,1) AND usiNr <= UPPER_BOUND(AY_XRELEASE,1) THEN
	(* No release if no more acknowledge *)
	IF AY_XRELEASE[usiNr] AND AY_XRELEASE[usiNr] = AY_XACKNOWLEDGEOLD[usiNr] AND NOT AY_XACKNOWLEDGE[usiNr] THEN
		AY_XRELEASE[usiNr] := FALSE;
	END_IF;	
	xRelease := AY_XRELEASE[usiNr] AND NOT xLockDown;
ELSE
	xRelease := FALSE;
END_IF;
IF usiNr >= LOWER_BOUND(AY_RRELEASE,1) AND usiNr <= UPPER_BOUND(AY_RRELEASE,1) THEN
	AY_RRELEASE[usiNr]	:= rNewRelease;
	rRelease 			:= AY_RRELEASE[usiNr];
ELSE
	rRelease := 0;
END_IF;

(* TIME *)
IF usiNr >= LOWER_BOUND(AY_RUN_TIME,1) AND usiNr <= UPPER_BOUND(AY_RUN_TIME,1) THEN
	AY_TON_RUN_TIME[usiNr](IN := NOT AY_TON_RUN_TIME[usiNr].Q AND xRelease AND xAcknowledge,
						   PT := T#1M);
	IF AY_TON_RUN_TIME[usiNr].Q THEN
		AY_RUN_TIME[usiNr] 			:= AY_RUN_TIME[usiNr] + 1;
		AY_RUN_TIME_TILL_ON[usiNr] 	:= AY_RUN_TIME_TILL_ON[usiNr] + 1;
	END_IF;
	IF NOT xRelease THEN
		AY_RUN_TIME_TILL_ON[usiNr] 	:= 0;
	END_IF;
END_IF;

scHz := scHzAll;
END_METHOD

METHOD GET_ENGINE_STATE : BOOL
VAR_INPUT
	usiNr			:	USINT;
END_VAR         	
VAR_OUTPUT	    	
	xAvaiable			:	BOOL;
	xRelease			:	BOOL;
	rRelease			:	REAL;
	xAcknowledge		:	BOOL;
	rAcknowledgeHz		:	REAL;
	xLockDown			:	BOOL;
	udiRunTime			:	UDINT;
	udiRunTimeTillOn	:	UDINT;
END_VAR
(* Avaiable *)
IF usiNr >= LOWER_BOUND(AY_XAVAIABLE,1) AND usiNr <= UPPER_BOUND(AY_XAVAIABLE,1) THEN
	xAvaiable := AY_XAVAIABLE[usiNr];
END_IF;

(* Release *)
IF usiNr >= LOWER_BOUND(AY_XRELEASE,1) AND usiNr <= UPPER_BOUND(AY_XRELEASE,1) THEN
	xRelease := AY_XRELEASE[usiNr];
END_IF;

(* Release *)
IF usiNr >= LOWER_BOUND(AY_RRELEASE,1) AND usiNr <= UPPER_BOUND(AY_RRELEASE,1) THEN
	rRelease := AY_RRELEASE[usiNr];
END_IF;

(* Acknowledge *)
IF usiNr >= LOWER_BOUND(AY_XACKNOWLEDGE,1) AND usiNr <= UPPER_BOUND(AY_XACKNOWLEDGE,1) THEN
	xAcknowledge := AY_XACKNOWLEDGE[usiNr];
END_IF;
IF usiNr >= LOWER_BOUND(AY_RACKNOWLEDGE,1) AND usiNr <= UPPER_BOUND(AY_RACKNOWLEDGE,1) THEN
	rAcknowledgeHz := AY_RACKNOWLEDGE[usiNr];
END_IF

(* LockDown *)
IF usiNr >= LOWER_BOUND(AY_LOCKDOWN,1) AND usiNr <= UPPER_BOUND(AY_LOCKDOWN,1) THEN
	xLockDown := AY_LOCKDOWN[usiNr];
END_IF;

(* Temp Min Run *)
IF usiNr >= LOWER_BOUND(AY_RUN_TIME,1) AND usiNr <= UPPER_BOUND(AY_RUN_TIME,1) THEN
	udiRunTime := AY_RUN_TIME[usiNr];
END_IF;

(* Temp Min Run Till On*)
IF usiNr >= LOWER_BOUND(AY_RUN_TIME_TILL_ON,1) AND usiNr <= UPPER_BOUND(AY_RUN_TIME_TILL_ON,1) THEN
	udiRunTimeTillOn := AY_RUN_TIME_TILL_ON[usiNr];
END_IF;
END_METHOD

METHOD RELEASE_ENGINE : BOOL
VAR_INPUT
	usiNr		:	USINT;
	xRelease	:	BOOL;
END_VAR
(* Release *)
IF usiNr >= LOWER_BOUND(AY_XRELEASE,1) AND usiNr <= UPPER_BOUND(AY_XRELEASE,1) THEN
	AY_XRELEASE[usiNr] := xRelease;
	IF NOT xRelease THEN
		AY_RRELEASE[usiNr] := 0;
	END_IF;
END_IF;
END_METHOD

PROPERTY LOWERBOUND : DINT
GET
LOWERBOUND := LOWER_BOUND(AY_XRELEASE,1);
END_GET
END_PROPERTY

PROPERTY UPPERBOUND : DINT
GET
UPPERBOUND := UPPER_BOUND(AY_XRELEASE,1);
END_GET
END_PROPERTY

METHOD SET_HZ_SCALE
VAR_INPUT
	scHz		:	CtaSysTypes.scHzParameter;
END_VAR
scHzAll := scHz;
END_METHOD

PROPERTY GET_ANZ_ENABLED : UINT
GET
VAR
	diForTemp	:	DINT;
END_VAR
GET_ANZ_ENABLED := 0;
FOR diForTemp := LOWER_BOUND(AY_XENABLED,1) TO UPPER_BOUND(AY_XENABLED,1) DO
	IF AY_XENABLED[diForTemp] THEN
		GET_ANZ_ENABLED := GET_ANZ_ENABLED + 1;
	END_IF;
END_FOR;
END_GET
END_PROPERTY

PROPERTY GET_SUM_ACKNOWLEDGE_HZ : REAL
GET
VAR
	diForTemp	:	DINT;
END_VAR
GET_SUM_ACKNOWLEDGE_HZ := 0;
FOR diForTemp := LOWER_BOUND(AY_RACKNOWLEDGE,1) TO UPPER_BOUND(AY_RACKNOWLEDGE,1) DO
	GET_SUM_ACKNOWLEDGE_HZ := GET_SUM_ACKNOWLEDGE_HZ + AY_RACKNOWLEDGE[diForTemp];
END_FOR;
END_GET
END_PROPERTY

END_FUNCTION_BLOCK

// 30 Program Organization Units/Group/GroupMember/Help/GROUPMEMBER
FUNCTION_BLOCK GROUPMEMBER
VAR_INPUT
	AY_MEMBER_OF		:	ARRAY[0..4] OF BOOL;
END_VAR
VAR_OUTPUT
	xTrigIsChanged		:	BOOL;
END_VAR
VAR
	AY_MEMBER_OF_OLD	:	ARRAY[0..4] OF BOOL;
	diFor1				:	DINT;
END_VAR

xTrigIsChanged := FALSE;
FOR diFor1 := LOWER_BOUND(AY_MEMBER_OF,1) TO UPPER_BOUND(AY_MEMBER_OF,1) DO
	IF AY_MEMBER_OF[diFor1] <> AY_MEMBER_OF_OLD[diFor1] THEN
		xTrigIsChanged 				:= TRUE;
		AY_MEMBER_OF_OLD[diFor1]	:= AY_MEMBER_OF[diFor1];
	END_IF
END_FOR;

END_FUNCTION_BLOCK

// 30 Program Organization Units/Group/GroupMember/Hydraulics/HYDRA
FUNCTION_BLOCK HYDRA EXTENDS GROUPBASE IMPLEMENTS ITF_HYDRA
VAR_OUTPUT
END_VAR
VAR
	xIsAddedToNessesary	:	BOOL;
	GROUPMEMBER			:	GROUPMEMBER;
END_VAR

SUPER^();
GROUPMEMBER();
IF GROUPMEMBER.xTrigIsChanged THEN
	xIsAddedToNessesary := FALSE;
END_IF;

METHOD MEMBER_OF : BOOL
VAR_INPUT
	usiGROUP_NR	: USINT;
END_VAR
IF usiGROUP_NR >= LOWER_BOUND(GROUPMEMBER.AY_MEMBER_OF,1) AND usiGROUP_NR <= UPPER_BOUND(GROUPMEMBER.AY_MEMBER_OF,1) THEN
	IF GROUPMEMBER.AY_MEMBER_OF[0] THEN
		MEMBER_OF := TRUE;
	ELSE
		MEMBER_OF := GROUPMEMBER.AY_MEMBER_OF[usiGROUP_NR];
	END_IF
ELSE
	MEMBER_OF := FALSE;
END_IF;
END_METHOD

//FB_Init ist immer implizit verfügbar und wird primär für die Initialisierung verwendet.
//Der Rückgabewert wird nicht ausgewertet. Für gezielte Einflussnahme können Sie
//die Methoden explizit deklarieren und darin mit dem Standard-Initialisierungscode 
//zusätzlichen Code bereitstellen. Sie können den Rückgabewert auswerten.
METHOD FB_Init: BOOL
VAR_INPUT    
bInitRetains: BOOL; // TRUE: Die Retain-Variablen werden initialisiert (Reset warm / Reset kalt)    
bInCopyCode: BOOL;  // TRUE: Die Instanz wird danach in den Kopiercode kopiert (Online-Change)
END_VAR
VAR_INPUT
	xAll	:	BOOL;
	xGp1	:	BOOL;
	xGp2	:	BOOL;
	xGp3	:	BOOL;
	xGp4	:	BOOL;
END_VAR
GROUPMEMBER.AY_MEMBER_OF[0] := xAll;
GROUPMEMBER.AY_MEMBER_OF[1] := xGp1;
GROUPMEMBER.AY_MEMBER_OF[2] := xGp2;
GROUPMEMBER.AY_MEMBER_OF[3]	:= xGp3;
GROUPMEMBER.AY_MEMBER_OF[4]	:= xGp4;
END_METHOD

END_FUNCTION_BLOCK

// 30 Program Organization Units/Manager/MANAGER
FUNCTION_BLOCK MANAGER IMPLEMENTS ITF_MANAGER
VAR_INPUT
    en_check                                        : INT;   						// Haupt-Check-State für die Engine-/Gruppenprüfung
    en_check_substate                               : INT;   						// Substate des Check-Prozesses
                                                                					
    xRelease                                        : BOOL;  						// BOOL-Trigger für eine Release-Anforderung
    iRelease                                        : INT;   						// Integer-Releasewert oder Release-Kommando
    rRelease                                        : REAL;  						// Realwert für Release-Parameter (z. B. Sollwert)
                                                                					
    en_release                                      : INT;   						// Haupt-State des Release-Vorgangs
    en_release_substate                             : INT;   						// Substate des Release-Vorgangs
    en_release_next                                 : INT;   						// Nächster Release-State (State-Machine)

    scHzRelease                                     : CtaSysTypes.scHzParameter;  	// Release-Parameter mit Hz-Information

    en_static_define_state_off                      : INT;   						// Definierter State für OFF-Zustand
	en_static_define_state_not_ready                : INT;   						// Definierter State für Nicht bereit-Zustand
    en_static_define_sub_state_off                  : INT;   						// Definierter Substate für OFF-Zustand
    en_static_define_lockdown                       : INT;   						// State für Lockdown-Bedingungen
    en_static_define_substate_check_new_state       : INT;   						// Substate zur Prüfung eines neuen State
    en_static_define_engine_release_from_substate   : INT;   						// Substate, wenn Engine in Release-ON gehen soll
	en_static_define_engine_release_off_substate    : INT;   						// Substate, wenn Engine in Release-OFF gehen soll
	en_static_define_state_ignore					: INT;							// Definierter State für ignorieren
END_VAR

VAR_OUTPUT
    iAvailable                                      : INT;   						// Verfügbarkeitskennzahl der Engine/Gruppe
    en_available                                    : INT;   						// Haupt-State der Verfügbarkeit
    en_available_substate                           : INT;   						// Substate der Verfügbarkeit
                                                             						
    iAcknowledged                                   : INT;   						// Integer-Wert zur Acknowledge-Verarbeitung
    rAcknowledgeHz                                  : REAL;  						// Realwert für Acknowledge-Hz
    en_acknowledge                                  : INT;   						// State für Acknowledge-Vorgang
    en_acknowledge_substate                         : INT;   						// Substate des Acknowledge-Vorgangs
                                                             						
    en_demand                                       : INT;   						// Haupt-State für Demand-/Anforderung
    en_demand_substate                              : INT;   						// Substate für Demand-/Anforderung
    
    ITF_MANAGER                                     : ITF_MANAGER; 					// Manager-Interface für Gruppen-/Engine-Steuerung
END_VAR

VAR
    sync_groups                                     : ARRAY[1..GVL_CONSTANT.MAX_GROUPS] OF DINT := [GVL_CONSTANT.MAX_GROUPS(1)];  // Array zur Synchronisationsverwaltung der Gruppen

    groups                                          : ARRAY[1..GVL_CONSTANT.MAX_GROUPS] OF ARRAY[0..40] OF ITF_GROUPBASE;         // Struktur aller Gruppen und ihrer Members

    groups_en_available                             : ARRAY[1..GVL_CONSTANT.MAX_GROUPS] OF INT; // Verfügbarkeits-State je Gruppe
    groups_en_available_substate                    : ARRAY[1..GVL_CONSTANT.MAX_GROUPS] OF INT; // Verfügbarkeits-Substate je Gruppe

    groups_engine_available                          : ARRAY[1..GVL_CONSTANT.MAX_GROUPS] OF INT; // Engine-Verfügbarkeitsstate je Gruppe

    groups_en_acknowledge                           : ARRAY[1..GVL_CONSTANT.MAX_GROUPS] OF INT; // Acknowledge-State je Gruppe
    groups_en_acknowledge_substate                  : ARRAY[1..GVL_CONSTANT.MAX_GROUPS] OF INT; // Acknowledge-Substate je Gruppe

    groups_engine_acknowledged                      : ARRAY[1..GVL_CONSTANT.MAX_GROUPS] OF INT; // Engine-Acknowledge-State je Gruppe
	groups_engine_released                       	: ARRAY[1..GVL_CONSTANT.MAX_GROUPS] OF INT; // Engine-Acknowledge-State je Gruppe

    groups_en_release                               : ARRAY[1..GVL_CONSTANT.MAX_GROUPS] OF INT; // Release-State je Gruppe
    groups_en_release_substate                  	: ARRAY[1..GVL_CONSTANT.MAX_GROUPS] OF INT; // release-Substate je Gruppe

	groups_en_demand								: ARRAY[1..GVL_CONSTANT.MAX_GROUPS] OF INT; // Demand-State je Gruppe

    AY_GROUPS_xReleaseCircuit                       : ARRAY[1..GVL_CONSTANT.MAX_GROUPS] OF BOOL; // Release-Freigabe je Circuit

    TEMP_ITF_GROUPBASE                              : ITF_GROUPBASE;  // Temp-Objekt für Gruppenoperationen
    TEMP_ITF_CIRCUIT                                : ITF_CIRCUIT;    // Temp-Circuit-Objekt
    TEMP_ITF_HYDRA                                  : ITF_HYDRA;      // Temp-Hydra-Objekt
    TEMP_ITF_HYDRA_MAX_CT                           : ITF_HYDRA;      // Temp-Hydra Objekt für max CT-Ermittlung

    diTempMemberCount                                : DINT;  // Temporäre Anzahl an Gruppenmitgliedern
    diFor1                                           : DINT;  // Schleifenzähler 1
    diFor2                                           : DINT;  // Schleifenzähler 2
    diFor3                                           : DINT;  // Schleifenzähler 3
    next_circuit_to_run_engine                       : DINT;  // Nächster Circuit, der gestartet werden soll
    next_engine_to_run                                : DINT;  // Nächste Engine, die starten soll
    next_circuit_to_stopp_engine                     : DINT;  // Nächster Circuit zum Ausschalten
    next_engine_to_stopp                             : DINT;  // Nächste Engine zum Ausschalten

    xTrigOn                                          : BOOL;  // Trigger für Start-/ON-Übergang
    xTrigOff                                         : BOOL;  // Trigger für Stop-/OFF-Übergang
    iTrigOffCount                                    : INT;   // Zähler für OFF-Triggerpflege
    iTrigOffMax                                      : INT;   // Maximal zulässige OFF-Triggerzeit

    en_check_old                                     : INT;   // Alter Check-State
	en_check_substate_old                            : INT;   // Alter Check-State
    en_release_old                                   : INT;   // Alter Release-State
	en_release_substate_old							 : INT;  // Alter Release-Substate
		
    uiCountGroupLockDown                             : UINT;  // Anzahl Gruppen im Lockdown
    uiCountEngineLockDown                            : UINT;  // Anzahl Engines im Lockdown
    uiCountEngineAcknowledge                         : UINT;  // Anzahl Engines, die Acknowledge benötigen
    uiCountGroupLockDownOld                          : UINT;  // Vorherige Lockdown-Gruppenzahl
    uiCountEngineAcknowledgeOld                      : UINT;  // Vorherige Anzahl Acknowledge-Engines
    uiCountEngineLockDownOld                         : UINT;  // Vorherige Lockdown-Enginezahl

	iAvailableTemp                                   : INT;   						// Verfügbarkeitskennzahl der Engine/Gruppe
	iAcknowledgedTemp                                : INT;   						// Integer-Wert zur Acknowledge-Verarbeitung
    iReleaseOld                                      : INT;   // Alter Releasewert
    iAcknowledgeOld                                  : INT;   // Alter Acknowledgewert
	rAcknowledgeTemp							     : REAL;
    xReleaseStopp                                    : BOOL;  // Stopp-Bedingung für Release
    TP_ReleaseLock                                   : Standard.TP;   // Timerbaustein für Release-Lock
	TP_ReleaseLockLockdown							 : Standard.TP;
    xResettReleaseLock_VIS                           : BOOL;  // Reset über VIS zum ReleaseLock

    lock_if_released_in_other_circuit                : BOOL;  // Lock, wenn Release in anderem Circuit aktiv ist

    // Parameter
    fbConfigFile                                     : CtaSysConfig.fbConfigFile; // Konfigurationsdatei-Handler
    scParameter                                      : scParameter;               // Parametrierobjekt

	priority_array									 : ARRAY[1..100] OF INT;
END_VAR

actParameter();

(* ITF *)
ITF_MANAGER := THIS^;

(* CHECK *)
CHECK();

(* AVAIABLE *)
AVAIABLE(); 

(* LOCKDOWN *)
LOCKDOWN();

(* ACKNOWLEDGE *)
ACKNOWLEDGE();

(* MANAGEMENT *)
ENGINE_MANAGEMENT();

(* RELEASE *)
RELEASE();

(* DEMAND *)
DEMAND();

(* UPDATE *)
UPDATE_AT_THE_END();

ACTION CHECK:
(* Set Check State *)
FOR diFor1 := LOWER_BOUND(groups,1) TO UPPER_BOUND(groups,1) DO
	set_check_of_group(groups[diFor1],en_check);
	set_check_substate_of_group(groups[diFor1],en_check_substate);
END_FOR;
END_ACTION

// Methode zum Setzen des Prüf-/Check-Status für alle relevanten Elemente einer Gruppe
METHOD set_check_of_group

VAR_INPUT
    // Array variabler Größe mit Objekten, die das Interface ITF_GROUPBASE implementieren
    _group : ARRAY[*] OF ITF_GROUPBASE;
    
    // Check-Zustand, der für alle relevanten Gruppenobjekte gesetzt werden soll
    _state : INT;
END_VAR

VAR
    // Laufvariable für die Iteration über das Gruppen-Array
    _diFor1 : DINT;
END_VAR
// Durchlaufe alle Elemente der ersten Dimension von _group
FOR _diFor1 := LOWER_BOUND(_group, 1) TO UPPER_BOUND(_group, 1) DO

    // Prüft, ob das aktuelle Array-Element das erwartete Interface unterstützt
    IF __QUERYINTERFACE(_group[_diFor1], _group[_diFor1]) THEN
        
        // Setzt den Check-Status des Elements anhand des übergebenen Zustands
        _group[_diFor1].set_check(_state);

    END_IF;
END_FOR;
END_METHOD

// Methode zum Setzen eines Sub-Check-/Sub-Status für alle relevanten Elemente einer Gruppe
METHOD set_check_substate_of_group

VAR_INPUT
    // Array variabler Größe mit Objekten, die das Interface ITF_GROUPBASE implementieren
    _group : ARRAY[*] OF ITF_GROUPBASE;
    
    // Sub-Check-/Sub-Status, der für alle relevanten Gruppenobjekte gesetzt werden soll
    _sub_state : INT;
END_VAR

VAR
    // Laufvariable für die Iteration über das Gruppen-Array
    _diFor1 : DINT;
END_VAR
// Durchlaufe alle Elemente der ersten Dimension des _group-Arrays
FOR _diFor1 := LOWER_BOUND(_group, 1) TO UPPER_BOUND(_group, 1) DO

    // Prüft, ob das aktuelle Element das erwartete Interface implementiert
    IF __QUERYINTERFACE(_group[_diFor1], _group[_diFor1]) THEN

        // Setzt den Sub-Check-/Sub-Status des Elements entsprechend dem übergebenen Wert
        _group[_diFor1].set_check_substate(_sub_state);
			
    END_IF;
END_FOR;
END_METHOD

METHOD get_next_engine_to_start 
VAR_INPUT
	enTYPE_OF_ENGINE_MANAGEMENT	:	TYPE_OF_ENGINE_MANAGEMENT;
END_VAR
VAR_OUTPUT
	next_circuit_to_start_engine  		: DINT;
	next_engine_to_start				: DINT;	
END_VAR
IF enTYPE_OF_ENGINE_MANAGEMENT = TYPE_OF_ENGINE_MANAGEMENT.RUN_1BY1 THEN
	engine_management_start_run_1_by_1(next_circuit_to_start_engine => next_circuit_to_start_engine,next_engine_to_start => next_engine_to_start);
(* EQUAL *)
ELSIF enTYPE_OF_ENGINE_MANAGEMENT = TYPE_OF_ENGINE_MANAGEMENT.RUN_EQUAL THEN
	engine_management_start_run_equal(next_circuit_to_start_engine => next_circuit_to_start_engine,next_engine_to_start => next_engine_to_start);
END_IF;
END_METHOD

METHOD get_next_engine_to_stopp 
VAR_INPUT
	enTYPE_OF_ENGINE_MANAGEMENT	:	TYPE_OF_ENGINE_MANAGEMENT;
END_VAR
VAR_OUTPUT
	next_circuit_to_stopp_engine  		: DINT;
	next_engine_to_stopp				: DINT;	
END_VAR

(* 1By1 *)
IF enTYPE_OF_ENGINE_MANAGEMENT = TYPE_OF_ENGINE_MANAGEMENT.RUN_1BY1 THEN
	engine_management_stopp_run_1_by_1(next_circuit_to_stopp_engine => next_circuit_to_stopp_engine,next_engine_to_stopp => next_engine_to_stopp);
(* EQUAL *)
ELSIF enTYPE_OF_ENGINE_MANAGEMENT = TYPE_OF_ENGINE_MANAGEMENT.RUN_EQUAL THEN
	engine_management_stopp_run_equal(next_circuit_to_stopp_engine => next_circuit_to_stopp_engine,next_engine_to_stopp => next_engine_to_stopp);	
END_IF;
END_METHOD

METHOD engine_management_start_run_1_by_1
VAR_OUTPUT
	next_circuit_to_start_engine  		: DINT;
	next_engine_to_start				: DINT;	
END_VAR
VAR 
	_xAvaiable							: BOOL;
	_xRelease							: BOOL;
	_rRelease							: REAL;
	_xAcknowledge						: BOOL;
	_rAcknowledge						: REAL;
	_xLockDown							: BOOL;
	_udiRunTime		    				: UDINT;
	_udiRunTimeTillOn   				: UDINT;
	_udiMinRunTime						: UDINT;
	_xIsAcknowledgeGroup				: BOOL;
END_VAR
(* Set Min Run Time To Max *)
_udiMinRunTime := 16#FFFFFFFF;
(* Set Lowest Acknowledge Group to False *)
_xIsAcknowledgeGroup := FALSE;
(* Set Circuit to 0 *)
next_circuit_to_start_engine := 0;
(* Set Engine to 0  *)
next_engine_to_start := 0;

FOR diFor1 := UPPER_BOUND(groups,1) TO LOWER_BOUND(groups,1) BY -1 DO 
	(* If No Error avaiable to release*)
	IF groups_en_acknowledge[diFor1] = en_release THEN		
		IF __QUERYINTERFACE(groups[diFor1][LOWER_BOUND(groups[diFor1],1)],TEMP_ITF_CIRCUIT) THEN
			IF TEMP_ITF_CIRCUIT.GET_ANZ_RELEASE > 0 AND TEMP_ITF_CIRCUIT.GET_ANZ_AVAIABLE > 0 THEN
				(* iterate Engine and Check if Avaiable and get the Minits *)
				FOR diFor2 := TEMP_ITF_CIRCUIT.UPPERBOUND TO TEMP_ITF_CIRCUIT.LOWERBOUND BY -1 DO
					TEMP_ITF_CIRCUIT.GET_ENGINE_STATE(	usiNr 			:= TO_USINT(diFor2),
														xAvaiable 		=> _xAvaiable,
														xRelease		=> _xRelease,
														rRelease		=> _rRelease,
														xAcknowledge 	=> _xAcknowledge,
														rAcknowledgeHz 	=> _rAcknowledge,
														xLockDown 		=> _xLockDown,
														udiRunTime 		=> _udiRunTime,
														udiRunTimeTillOn=> _udiRunTimeTillOn);
					(* Get time if Avaiable *)
					IF _xAvaiable AND NOT _xRelease AND NOT _xLockDown THEN
						IF _udiRunTime <= _udiMinRunTime THEN
							_udiMinRunTime 					:= _udiRunTime;
							next_circuit_to_start_engine 	:= diFor1;
							next_engine_to_start  			:= diFor2;
						END_IF;			
					END_IF;						
				END_FOR;
			END_IF;
		END_IF;
	END_IF;
END_FOR;
(* Get new Ccuit if not possible to add ad running circuti *)
IF next_circuit_to_start_engine = 0 AND next_engine_to_start = 0  THEN
	FOR diFor1 := UPPER_BOUND(groups,1) TO LOWER_BOUND(groups,1) BY -1 DO
		(* If No Error avaiable to release*)
		IF groups_en_available[diFor1] = en_release OR groups_en_acknowledge[diFor1] = en_release THEN	
			IF __QUERYINTERFACE(groups[diFor1][LOWER_BOUND(groups[diFor1],1)],TEMP_ITF_CIRCUIT) THEN
				IF TEMP_ITF_CIRCUIT.GET_ANZ_AVAIABLE > 0 THEN
					(* iterate Engine and Check if Avaiable and get the Minits *)
					FOR diFor2 := TEMP_ITF_CIRCUIT.UPPERBOUND TO TEMP_ITF_CIRCUIT.LOWERBOUND BY -1 DO
						TEMP_ITF_CIRCUIT.GET_ENGINE_STATE(	usiNr 			:= TO_USINT(diFor2),
															xAvaiable 		=> _xAvaiable,
															xRelease		=> _xRelease,
															rRelease		=> _rRelease,
															xAcknowledge 	=> _xAcknowledge,
															rAcknowledgeHz 	=> _rAcknowledge,
															xLockDown 		=> _xLockDown,
															udiRunTime 		=> _udiRunTime,
															udiRunTimeTillOn=> _udiRunTimeTillOn);
						(* Get time if Avaiable *)
						IF _xAvaiable AND NOT _xRelease AND NOT _xLockDown THEN
							IF _udiRunTime <= _udiMinRunTime AND (NOT _xIsAcknowledgeGroup OR groups_en_acknowledge[diFor1] = en_release) THEN
								_xIsAcknowledgeGroup			:= groups_en_acknowledge[diFor1] = en_release;
								_udiMinRunTime 					:= _udiRunTime;
								next_circuit_to_start_engine 	:= diFor1;
								next_engine_to_start  			:= diFor2;
							END_IF;			
						END_IF;						
					END_FOR;
				END_IF;
			END_IF;
		END_IF;
	END_FOR;		
END_IF;
END_METHOD

METHOD engine_management_start_run_equal
VAR_OUTPUT
	next_circuit_to_start_engine  		: DINT;
	next_engine_to_start				: DINT;	
END_VAR
VAR 
	_xAvaiable							: BOOL;
	_xRelease							: BOOL;
	_rRelease							: REAL;
	_xAcknowledge						: BOOL;
	_rAcknowledge						: REAL;
	_xLockDown							: BOOL;
	_udiRunTime		    				: UDINT;
	_udiRunTimeTillOn   				: UDINT;
	_udiMinRunTime						: UDINT;
	_uiLowestWorkloadCircuit			: UINT;
END_VAR
(* Set Min Run Time To Max *)
_udiMinRunTime := 16#FFFFFFFF;
(* Set Lowest Workload Circuit to MAX *)
_uiLowestWorkloadCircuit := 16#FFFF;
(* Set Circuit to 0 *)
next_circuit_to_start_engine := 0;
(* Set Engine to 0  *)
next_engine_to_start := 0;
FOR diFor1 := UPPER_BOUND(groups,1) TO LOWER_BOUND(groups,1) BY -1 DO 
	(* If No Error avaiable to release*)
	IF groups_en_available[diFor1] = en_release  OR groups_en_acknowledge[diFor1] = en_release THEN	
		IF __QUERYINTERFACE(groups[diFor1][LOWER_BOUND(groups[diFor1],1)],TEMP_ITF_CIRCUIT) THEN
			IF TEMP_ITF_CIRCUIT.GET_ANZ_RELEASE <= _uiLowestWorkloadCircuit AND TEMP_ITF_CIRCUIT.GET_ANZ_AVAIABLE > 0 THEN
				_uiLowestWorkloadCircuit := TEMP_ITF_CIRCUIT.GET_ANZ_RELEASE; 
				(* iterate Engine and Check if Avaiable and get the Minits *)
				FOR diFor2 := TEMP_ITF_CIRCUIT.UPPERBOUND TO TEMP_ITF_CIRCUIT.LOWERBOUND BY -1 DO
					TEMP_ITF_CIRCUIT.GET_ENGINE_STATE(	usiNr 			:= TO_USINT(diFor2),
														xAvaiable 		=> _xAvaiable,
														xRelease		=> _xRelease,
														rRelease		=> _rRelease,
														xAcknowledge 	=> _xAcknowledge,
														rAcknowledgeHz 	=> _rAcknowledge,
														xLockDown 		=> _xLockDown,
														udiRunTime 		=> _udiRunTime,
														udiRunTimeTillOn=> _udiRunTimeTillOn);
					(* Get time if Avaiable *)
					IF _xAvaiable AND NOT _xRelease AND NOT _xLockDown THEN
						IF _udiRunTime <= _udiMinRunTime THEN
							_udiMinRunTime 					:= _udiRunTime;
							next_circuit_to_start_engine 	:= diFor1;
							next_engine_to_start  			:= diFor2;
						END_IF;			
					END_IF;						
				END_FOR;
			END_IF;
		END_IF;
	END_IF;
END_FOR;
END_METHOD

METHOD engine_management_stopp_run_1_by_1
VAR_OUTPUT
	next_circuit_to_stopp_engine  		: DINT;
	next_engine_to_stopp				: DINT;	
END_VAR
VAR 
	_xAvaiable							: BOOL;
	_xRelease							: BOOL;
	_rRelease							: REAL;
	_xAcknowledge						: BOOL;
	_rAcknowledge						: REAL;
	_xLockDown							: BOOL;
	_udiRunTime		    				: UDINT;
	_udiRunTimeTillOn   				: UDINT;
	_udiMaxRunTimeTillOn				: UDINT;
	_uiHighestWorkloadCircuit			: UINT;
	_uiLowestWorkloadCircuit			: UINT;
END_VAR
(* Set Highest Workload Circuit to Min *)
_uiHighestWorkloadCircuit := 16#0000;
(* Set Lowest Workload Circuit to MAX *)
_uiLowestWorkloadCircuit := 16#FFFF;
(* Set Max Run Time To Min *)
_udiMaxRunTimeTillOn := 16#0000;
(* Set Circuit to 0 *)
next_circuit_to_stopp_engine := 0;

(* Set Engine to 0  *)
next_engine_to_stopp := 0;

FOR diFor1 := UPPER_BOUND(groups,1) TO LOWER_BOUND(groups,1) BY -1 DO 
	(* If No Error avaiable to release*)
	IF groups_en_acknowledge[diFor1] = en_release THEN	
		IF __QUERYINTERFACE(groups[diFor1][LOWER_BOUND(groups[diFor1],1)],TEMP_ITF_CIRCUIT) THEN
			IF TEMP_ITF_CIRCUIT.GET_ANZ_RELEASE > 0 THEN
				IF TEMP_ITF_CIRCUIT.GET_ANZ_RELEASE <= _uiLowestWorkloadCircuit THEN
					IF TEMP_ITF_CIRCUIT.GET_ANZ_RELEASE < _uiLowestWorkloadCircuit THEN
						_uiLowestWorkloadCircuit := TEMP_ITF_CIRCUIT.GET_ANZ_RELEASE; 
						(* Set Max Run Time To Min *)
						_udiMaxRunTimeTillOn := 16#0000;
					END_IF;

					(* iterate Engine and Check if Avaiable and get the Minits *)
					FOR diFor2 := TEMP_ITF_CIRCUIT.UPPERBOUND TO TEMP_ITF_CIRCUIT.LOWERBOUND BY -1 DO
						TEMP_ITF_CIRCUIT.GET_ENGINE_STATE(	usiNr 			:= TO_USINT(diFor2),
															xAvaiable 		=> _xAvaiable,
															xRelease		=> _xRelease,
															rRelease		=> _rRelease,
															xAcknowledge 	=> _xAcknowledge,
															rAcknowledgeHz 	=> _rAcknowledge,
															xLockDown 		=> _xLockDown,
															udiRunTime 		=> _udiRunTime,
															udiRunTimeTillOn=> _udiRunTimeTillOn);
						(* Get time if Running *)
						IF _xRelease THEN
							IF _udiRunTimeTillOn >= _udiMaxRunTimeTillOn THEN
								_udiMaxRunTimeTillOn 			:= _udiRunTimeTillOn;
								next_circuit_to_stopp_engine 	:= diFor1;
								next_engine_to_stopp 			:= diFor2;
							END_IF;			
						END_IF;						
					END_FOR;
				END_IF;
			END_IF;
		END_IF;
	END_IF;
END_FOR;
END_METHOD

METHOD engine_management_stopp_run_equal
VAR_OUTPUT
	next_circuit_to_stopp_engine  		: DINT;
	next_engine_to_stopp				: DINT;	
END_VAR
VAR 
	_xAvaiable							: BOOL;
	_xRelease							: BOOL;
	_rRelease							: REAL;
	_xAcknowledge						: BOOL;
	_rAcknowledge						: REAL;
	_xLockDown							: BOOL;
	_udiRunTime		    				: UDINT;
	_udiRunTimeTillOn   				: UDINT;
	_udiMaxRunTimeTillOn				: UDINT;
	_uiHighestWorkloadCircuit			: UINT;
	_uiLowestWorkloadCircuit			: UINT;
END_VAR
(* Set Highest Workload Circuit to Min *)
_uiHighestWorkloadCircuit := 16#0000;
(* Set Lowest Workload Circuit to MAX *)
_uiLowestWorkloadCircuit := 16#FFFF;
(* Set Max Run Time To Min *)
_udiMaxRunTimeTillOn := 16#0000;
(* Set Circuit to 0 *)
next_circuit_to_stopp_engine := 0;

(* Set Engine to 0  *)
next_engine_to_stopp := 0;


FOR diFor1 := UPPER_BOUND(groups,1) TO LOWER_BOUND(groups,1) BY -1 DO 
	(* If No Error avaiable to release*)
	IF groups_en_available[diFor1] = en_release OR groups_en_acknowledge[diFor1] = en_release THEN	
		IF __QUERYINTERFACE(groups[diFor1][LOWER_BOUND(groups[diFor1],1)],TEMP_ITF_CIRCUIT) THEN
			IF TEMP_ITF_CIRCUIT.GET_ANZ_RELEASE >= _uiHighestWorkloadCircuit THEN
				IF TEMP_ITF_CIRCUIT.GET_ANZ_RELEASE > _uiHighestWorkloadCircuit THEN
					_uiHighestWorkloadCircuit := TEMP_ITF_CIRCUIT.GET_ANZ_RELEASE; 
					(* Set Max Run Time To Min *)
					_udiMaxRunTimeTillOn := 16#0000;				
				END_IF;
				(* iterate Engine and Check if Avaiable and get the time *)
				FOR diFor2 := TEMP_ITF_CIRCUIT.UPPERBOUND TO TEMP_ITF_CIRCUIT.LOWERBOUND BY -1 DO
					TEMP_ITF_CIRCUIT.GET_ENGINE_STATE(	usiNr 			:= TO_USINT(diFor2),
														xAvaiable 		=> _xAvaiable,
														xRelease		=> _xRelease,
														rRelease		=> _rRelease,
														xAcknowledge 	=> _xAcknowledge,
														rAcknowledgeHz 	=> _rAcknowledge,
														xLockDown 		=> _xLockDown,
														udiRunTime 		=> _udiRunTime,
														udiRunTimeTillOn=> _udiRunTimeTillOn);
					(* Get time if Running *)
					IF _xRelease THEN
						IF _udiRunTimeTillOn >= _udiMaxRunTimeTillOn THEN
							_udiMaxRunTimeTillOn 			:= _udiRunTimeTillOn;
							next_circuit_to_stopp_engine 	:= diFor1;
							next_engine_to_stopp 			:= diFor2;
						END_IF;			
					END_IF;						
				END_FOR;
			END_IF;
		END_IF;
	END_IF;
END_FOR;
END_METHOD

ACTION ENGINE_MANAGEMENT:
(* ------------------------------------------------------------- *)
(* Engine Trigger Logic: TRIG ON / TRIG OFF and Release Handling   *)
(* ------------------------------------------------------------- *)

(* Wait until no TRIG ON is active, then determine next engine to run *)
IF NOT xTrigOn THEN
    get_next_engine_to_start(	enTYPE_OF_ENGINE_MANAGEMENT 	:= scParameter.fbiTypeOfEngineManagement.proValue,
        						next_circuit_to_start_engine 	=> next_circuit_to_run_engine,
        						next_engine_to_start  			=> next_engine_to_run);
END_IF;

(* Wait until no TRIG OFF is active, then determine next engine to stop *)
IF NOT xTrigOff THEN
    get_next_engine_to_stopp(	enTYPE_OF_ENGINE_MANAGEMENT 	:= scParameter.fbiTypeOfEngineManagement.proValue,
        						next_circuit_to_stopp_engine 	=> next_circuit_to_stopp_engine,
        						next_engine_to_stopp  			=> next_engine_to_stopp );
END_IF;

(* Check if engine is available and TRIG ON conditions are met *)
IF next_circuit_to_run_engine > 0 AND next_engine_to_run > 0 THEN
    IF xRelease AND iRelease > 0 THEN
		IF en_check = en_release THEN
			(* Handle group lockdown events *)
			IF uiCountGroupLockDown > uiCountGroupLockDownOld AND (en_available <> en_static_define_lockdown OR en_acknowledge <> en_static_define_lockdown) AND NOT xReleaseStopp AND NOT TP_ReleaseLockLockdown.Q THEN
				xTrigOn := TRUE;
				TP_ReleaseLock(IN	:= FALSE ,PT := T#0S);
				xReleaseStopp := TRUE;
			(* Handle engine lockdown events *)
			ELSIF uiCountEngineLockDown > uiCountEngineLockDownOld AND (en_available <> en_static_define_lockdown OR en_acknowledge <> en_static_define_lockdown) AND NOT xReleaseStopp AND NOT TP_ReleaseLockLockdown.Q THEN
				xTrigOn := TRUE;
				TP_ReleaseLock(IN	:= FALSE ,PT := T#0S);
				xReleaseStopp := TRUE;
			(* Handle engine turning off unexpectedly *)
			ELSIF uiCountEngineAcknowledge < uiCountEngineAcknowledgeOld AND iRelease > TO_INT(uiCountEngineAcknowledge) AND (en_available <> en_static_define_lockdown OR en_acknowledge <> en_static_define_lockdown) AND NOT xReleaseStopp AND NOT TP_ReleaseLockLockdown.Q THEN
				xTrigOn := TRUE;
				TP_ReleaseLock(IN	:= FALSE ,PT := T#0S);
				xReleaseStopp := TRUE;
			(* Normal case: Add engine if release request exceeds acknowledge and no lock active *)
			ELSIF iRelease > iAcknowledged AND NOT TP_ReleaseLock.Q AND NOT xTrigOn AND NOT xReleaseStopp THEN
				TP_ReleaseLock(IN := FALSE); (* Reset pulse before trigger *)
				xTrigOn := TRUE;
				xReleaseStopp := TRUE;
			END_IF;
		END_IF;
    ELSE
        xTrigOn := FALSE; (* Release not active → no TRIG ON *)
    END_IF;
ELSIF en_acknowledge = en_static_define_lockdown THEN
	TP_ReleaseLock(IN	:= FALSE ,PT := T#0S);
END_IF;

TP_ReleaseLockLockdown(IN := xReleaseStopp,PT := T#5S);

(* Manage normal release lock timer with minimum of 60s *)
IF NOT xResettReleaseLock_VIS AND xRelease THEN
    IF scParameter.fbtZuschaltSperrzeit.proValue > T#60S THEN
        TP_ReleaseLock(PT := scParameter.fbtZuschaltSperrzeit.proValue);
    ELSE
        TP_ReleaseLock(PT := T#60S);
    END_IF;
ELSE
    TP_ReleaseLock(IN := FALSE, PT := T#0MS);
    xResettReleaseLock_VIS := FALSE;
END_IF;

(* Check if engine is available and TRIG OFF conditions are met *)
IF next_circuit_to_stopp_engine > 0 AND next_engine_to_stopp > 0 THEN
    IF xRelease THEN
        (* Reset case: Release equals acknowledge → reset counters *)
        IF iRelease = iAcknowledged THEN
            iTrigOffMax := 0;
            iTrigOffCount := 0;
            IF xTrigOn THEN (* Prevent endless engine running *)
                xTrigOn := FALSE;
                xTrigOff := TRUE;
                next_circuit_to_stopp_engine := next_circuit_to_run_engine;
                next_engine_to_stopp  := next_engine_to_run;
            END_IF

        (* Normal reduction: Release < acknowledge → trigger engine off *)
        ELSIF iRelease < iAcknowledged THEN
            IF iRelease < iReleaseOld OR iAcknowledged > iAcknowledgeOld THEN
                iTrigOffMax := MIN(iAcknowledged, iTrigOffMax + iReleaseOld - iRelease);
            END_IF
            IF iTrigOffCount < iTrigOffMax THEN
                iTrigOffCount := iTrigOffCount + 1;
                xTrigOff := TRUE;
            END_IF;
        END_IF;

    ELSE
        xTrigOff := FALSE; (* Release inactive → no TRIG OFF *)
    END_IF;
END_IF;

(* Set Release array and trigger engines accordingly *)
FOR diFor1 := LOWER_BOUND(groups,1) TO UPPER_BOUND(groups,1) DO
    IF __QUERYINTERFACE(groups[diFor1][LOWER_BOUND(groups[diFor1],1)], TEMP_ITF_CIRCUIT) THEN
        IF groups_en_acknowledge[diFor1] <> en_static_define_lockdown OR groups_en_available[diFor1] = en_release OR groups_en_available[diFor1] = en_release_next THEN
			(* Stop engine if it is next to be turned off *)
			IF diFor1 = next_circuit_to_stopp_engine AND xTrigOff THEN
				TEMP_ITF_CIRCUIT.RELEASE_ENGINE(TO_USINT(next_engine_to_stopp), FALSE);
				xTrigOff := FALSE;
				xTrigOn := FALSE;
			END_IF;			
            IF TEMP_ITF_CIRCUIT.IS_RELEVANT_TO_RELEASE THEN
                (* Release engine if it is next to run and TRIG ON is active *)
                IF (groups_en_available[diFor1] 	= en_release 		OR 
					groups_en_available[diFor1] 	= en_release_next 	OR 
					groups_en_acknowledge[diFor1] 	= en_release	) 	AND 
					diFor1 = next_circuit_to_run_engine 				AND 
					xTrigOn 											AND 
					iRelease > 0 										THEN
                    groups_en_release[diFor1] := en_release;
					groups_en_release_substate[diFor1] 	:= en_release_substate;
                    IF groups_en_acknowledge_substate[diFor1] >= en_static_define_engine_release_from_substate AND groups_en_acknowledge_substate[diFor1] <= en_static_define_engine_release_off_substate THEN
                        IF TEMP_ITF_CIRCUIT.IS_RELEVANT_TO_RELEASE AND AY_GROUPS_xReleaseCircuit[diFor1] THEN
							TEMP_ITF_CIRCUIT.RELEASE_ENGINE(TO_USINT(next_engine_to_run), TRUE);
							xTrigOn := FALSE;
                        	TP_ReleaseLock(IN := TRUE);
						END_IF;
                    ELSE
                        TEMP_ITF_CIRCUIT.ALL_OFF();
                    END_IF;
                ELSIF groups_en_release[diFor1] = en_release AND groups_en_acknowledge_substate[diFor1] < en_static_define_engine_release_from_substate OR groups_en_acknowledge_substate[diFor1] > en_static_define_engine_release_off_substate THEN
                    TEMP_ITF_CIRCUIT.ALL_OFF();
					groups_en_release[diFor1] 			:= en_release;
					groups_en_release_substate[diFor1] 	:= en_release_substate;	
				ELSIF groups_en_release[diFor1] = en_release AND (TEMP_ITF_CIRCUIT.GET_ANZ_RELEASE = 0 OR iRelease = 0) THEN
					groups_en_release[diFor1] 			:= en_static_define_state_off;
					groups_en_release_substate[diFor1] 	:= en_static_define_sub_state_off;	
				ELSIF NOT xRelease THEN
					TEMP_ITF_CIRCUIT.ALL_OFF();
					groups_en_release[diFor1] 			:= en_release;
					groups_en_release_substate[diFor1] 	:= en_release_substate;				
                END_IF;
            ELSE
                TEMP_ITF_CIRCUIT.ALL_OFF();
				groups_en_release[diFor1] 			:= en_release;
				groups_en_release_substate[diFor1] 	:= en_release_substate;
            END_IF;
        ELSE
            TEMP_ITF_CIRCUIT.ALL_OFF();
			groups_en_release[diFor1] 			:= en_static_define_lockdown;
			groups_en_release_substate[diFor1] 	:= en_static_define_sub_state_off;
        END_IF;
		groups_engine_released[diFor1] := TO_INT( TEMP_ITF_CIRCUIT.GET_ANZ_RELEASE);
    ELSE
        groups_en_release[diFor1] 			:= en_static_define_state_off;
		groups_en_release_substate[diFor1] 	:= en_static_define_sub_state_off;
    END_IF;
END_FOR;

(* Apply HZ scale to relevant circuits *)
FOR diFor1 := LOWER_BOUND(groups,1) TO UPPER_BOUND(groups,1) DO
    IF __QUERYINTERFACE(groups[diFor1][LOWER_BOUND(groups[diFor1],1)], TEMP_ITF_CIRCUIT) THEN
        IF TEMP_ITF_CIRCUIT.IS_RELEVANT_TO_RELEASE THEN
            TEMP_ITF_CIRCUIT.SET_HZ_SCALE(scHzRelease);
        END_IF;
    END_IF;
END_FOR;

(* Set cyclic speed proportionally if acknowledge has not changed *)
IF iAcknowledged = iAcknowledgeOld THEN
    FOR diFor1 := LOWER_BOUND(groups,1) TO UPPER_BOUND(groups,1) DO
        IF __QUERYINTERFACE(groups[diFor1][LOWER_BOUND(groups[diFor1],1)], TEMP_ITF_CIRCUIT) THEN
            IF TEMP_ITF_CIRCUIT.IS_RELEVANT_TO_RELEASE THEN
            	TEMP_ITF_CIRCUIT.prorRelease := rRelease;
            END_IF;
        END_IF;
    END_FOR;
END_IF;
END_ACTION

ACTION UPDATE_AT_THE_END:
en_release_old 				:= en_release;
en_release_substate_old 	:= en_release_substate;
en_check_old				:= en_check;
en_check_substate_old		:= en_check_substate;

iReleaseOld					:= iRelease;
uiCountEngineAcknowledgeOld := uiCountEngineAcknowledge;
uiCountEngineLockDownOld 	:= uiCountEngineLockDown;
uiCountGroupLockDownOld		:= uiCountGroupLockDown;
xReleaseStopp 				:= FALSE;
END_ACTION

ACTION ACKNOWLEDGE:
IF en_release = en_release_old THEN
	iAcknowledgeOld 			:= iAcknowledged;
	iAcknowledgedTemp 			:= 0;
	rAcknowledgeTemp			:= 0;
	FOR diFor1 := LOWER_BOUND(groups,1) TO UPPER_BOUND(groups,1) DO
		// Prüfen, ob Gruppe ein gültiges Circuit-Interface hat
		IF __QUERYINTERFACE(groups[diFor1][0], TEMP_ITF_CIRCUIT) THEN
	
			// Tatsächlichen Acknowledge-Status ermitteln
			IF groups_en_release[diFor1] = en_release THEN
				groups_en_acknowledge[diFor1] := check_acknowledge_of_group(diFor1, groups[diFor1], groups_en_release[diFor1]);
				groups_en_acknowledge_substate[diFor1] := check_acknowledge_substate_of_group(diFor1, groups[diFor1], groups_en_release_substate[diFor1]);
			ELSE
				groups_en_acknowledge[diFor1] := groups_en_release[diFor1];
				groups_en_acknowledge_substate[diFor1] := groups_en_release_substate[diFor1];			
			END_IF
	
			// Anzahl der acknowledged Engines ermitteln
			groups_engine_acknowledged[diFor1] := TO_INT(TEMP_ITF_CIRCUIT.GET_ANZ_ACKNOWLEDGE);
			iAcknowledgedTemp := iAcknowledgedTemp + groups_engine_acknowledged[diFor1];
			rAcknowledgeTemp  := rAcknowledgeTemp + TEMP_ITF_CIRCUIT.GET_SUM_ACKNOWLEDGE_HZ;
		ELSE
			// Keine Engines verfügbar
			groups_en_acknowledge[diFor1] := en_static_define_lockdown;
			groups_en_acknowledge_substate[diFor1] := en_static_define_sub_state_off;
			groups_engine_acknowledged[diFor1] := 0;
		END_IF;
	END_FOR;
	// Wert setzen
	iAcknowledged := iAcknowledgedTemp;
	rAcknowledgeHz := rAcknowledgeTemp;
	uiCountEngineAcknowledge := TO_UINT(iAcknowledged);	
	// Manager Acknowledge aggregieren
	en_acknowledge 				:= en_static_define_lockdown;
	en_acknowledge_substate 	:= en_static_define_sub_state_off;
	FOR diFor1 := LOWER_BOUND(groups_en_acknowledge,1) TO UPPER_BOUND(groups_en_acknowledge,1) DO
		IF groups_en_acknowledge[diFor1] = en_release THEN
			en_acknowledge := groups_en_acknowledge[diFor1];
			IF groups_en_acknowledge_substate[diFor1] = en_release_substate THEN
				en_acknowledge_substate := groups_en_acknowledge_substate[diFor1];
				RETURN;
			ELSIF groups_en_acknowledge_substate[diFor1] = en_release_substate_old THEN
				en_acknowledge_substate := groups_en_acknowledge_substate[diFor1];
				RETURN;
			ELSE
				en_acknowledge_substate := groups_en_acknowledge_substate[diFor1];
			END_IF;
		END_IF;
	END_FOR;
	FOR diFor1 := LOWER_BOUND(groups_en_acknowledge_substate,1) TO UPPER_BOUND(groups_en_acknowledge_substate,1) DO
		IF groups_en_acknowledge_substate[diFor1] > en_acknowledge_substate AND groups_en_acknowledge[diFor1] = en_release THEN
			en_acknowledge := groups_en_acknowledge[diFor1];
			en_acknowledge_substate := groups_en_acknowledge_substate[diFor1];
			RETURN;
		END_IF;
	END_FOR
	IF en_acknowledge = en_release THEN
		RETURN;
	END_IF;
	FOR diFor1 := LOWER_BOUND(groups_en_acknowledge,1) TO UPPER_BOUND(groups_en_acknowledge,1) DO
		IF groups_en_release[diFor1] = en_release THEN
			en_acknowledge 				:= groups_en_release[diFor1];
			en_acknowledge_substate 	:= groups_en_acknowledge_substate[diFor1];
			RETURN;
		END_IF;
	END_FOR;
	FOR diFor1 := LOWER_BOUND(groups_en_acknowledge,1) TO UPPER_BOUND(groups_en_acknowledge,1) DO
		IF groups_en_release[diFor1] = en_release_old THEN
			en_acknowledge 				:= groups_en_release[diFor1];
			en_acknowledge_substate 	:= groups_en_acknowledge_substate[diFor1];
			RETURN;	
		END_IF;
	END_FOR;
	FOR diFor1 := LOWER_BOUND(groups_en_acknowledge,1) TO UPPER_BOUND(groups_en_acknowledge,1) DO
		IF groups_en_acknowledge[diFor1] = en_release_old THEN
			en_acknowledge 				:= groups_en_acknowledge[diFor1];
			en_acknowledge_substate 	:= groups_en_acknowledge_substate[diFor1];	
			RETURN;
		END_IF;
	END_FOR;
	FOR diFor1 := LOWER_BOUND(groups_en_acknowledge,1) TO UPPER_BOUND(groups_en_acknowledge,1) DO	
		IF groups_en_acknowledge[diFor1] = en_static_define_lockdown THEN
			en_acknowledge 				:= groups_en_acknowledge[diFor1];
			en_acknowledge_substate 	:= groups_en_acknowledge_substate[diFor1];			
		END_IF;
	END_FOR
END_IF;
END_ACTION

(* Methode, die den Acknowledge-Zustand aller Mitglieder einer Gruppe überprüft und den Status der Gruppe zurückgibt *)
METHOD check_acknowledge_of_group : INT
VAR_INPUT
	_group_nr			 : DINT;	// Gruppennummer als Info
    (* Eingabeparameter: Eine Array von Gruppenmitgliedern (Interface vom Typ ITF_GROUPBASE) *)
    _group               : ARRAY[*] OF ITF_GROUPBASE;
    
    (* Eingabeparameter: Der erwartete Acknowledge-Zustand, auf den alle Mitglieder überprüft werden *)
    _expectet_state      : INT;
END_VAR

VAR
    (* Interne Variable für die Schleifenindizierung *)
    _diFor1              : DINT;

END_VAR
(* Initialisierung des Check-Status der Gruppe auf "Lockdown" *)
check_acknowledge_of_group := en_static_define_lockdown;

(* Iteration durch alle Mitglieder der Gruppe, um den erwarteten Zustand zu überprüfen *)
FOR _diFor1 := LOWER_BOUND(_group, 1) TO UPPER_BOUND(_group, 1) DO
    (* Prüfen, ob das aktuelle Element in der Gruppe ein gültiges Interface hat *)
    IF __QUERYINTERFACE(_group[_diFor1], _group[_diFor1]) THEN
        (* Wenn das Interface gültig ist, setze den Check-Status auf den erwarteten Zustand *)
        check_acknowledge_of_group := _expectet_state;
    END_IF;
END_FOR;

(* Iteration durch alle Mitglieder der Gruppe, um den Zustand jedes Mitglieds zu überprüfen und den Gruppenstatus anzupassen *)
FOR _diFor1 := LOWER_BOUND(_group, 1) TO UPPER_BOUND(_group, 1) DO
    (* Wieder prüfen, ob das aktuelle Element in der Gruppe ein gültiges Interface hat *)
    IF __QUERYINTERFACE(_group[_diFor1], _group[_diFor1]) THEN
        (* Überprüfen, ob das Mitglied für das Acknowledge relevant ist (d.h., ob es nicht ignoriert wird) *)
        IF NOT _group[_diFor1].IS_NOT_RELEVANT_TO_ACKNOWLEDGE THEN
            (* Wenn das Acknowledge des Mitglieds nicht dem erwarteten Zustand entspricht *)
            IF _group[_diFor1].acknowledge <> _expectet_state THEN
                (* Wenn der Zustand nicht dem erwarteten Zustand entspricht, setze den Gruppen-Check-Status auf den tatsächlichen Acknowledge-Wert des Mitglieds *)
                check_acknowledge_of_group := _group[_diFor1].acknowledge;
            	IF check_acknowledge_of_group = en_static_define_lockdown THEN
					EXIT;
				END_IF;
			END_IF;
        END_IF;
    END_IF;
END_FOR;
END_METHOD

(* Methode, die den Acknowledge-Zustand aller Mitglieder einer Gruppe überprüft und den Status der Gruppe zurückgibt *)
METHOD check_acknowledge_substate_of_group : INT
VAR_INPUT
	_group_nr			 : DINT;	// Gruppennummer als Info
    (* Eingabeparameter: Eine Array von Gruppenmitgliedern (Interface vom Typ ITF_GROUPBASE) *)
    _group               : ARRAY[*] OF ITF_GROUPBASE;
    
    (* Eingabeparameter: Der erwartete Acknowledge-Zustand, auf den alle Mitglieder überprüft werden *)
    _expectet_substate   : INT;
END_VAR

VAR
    (* Interne Variable für die Schleifenindizierung *)
    _diFor1              : DINT;
END_VAR
(* Initialisierung des Check-Status der Gruppe auf "Lockdown" *)
check_acknowledge_substate_of_group := en_static_define_sub_state_off;

(* Iteration durch alle Mitglieder der Gruppe, um den erwarteten Zustand zu überprüfen *)
FOR _diFor1 := LOWER_BOUND(_group, 1) TO UPPER_BOUND(_group, 1) DO
    (* Prüfen, ob das aktuelle Element in der Gruppe ein gültiges Interface hat *)
    IF __QUERYINTERFACE(_group[_diFor1], _group[_diFor1]) THEN
        (* Wenn das Interface gültig ist, setze den Check-Status auf den erwarteten Zustand *)
        check_acknowledge_substate_of_group := _expectet_substate;
    END_IF;
END_FOR;

(* Iteration durch alle Mitglieder der Gruppe, um den Zustand jedes Mitglieds zu überprüfen und den Gruppenstatus anzupassen *)
FOR _diFor1 := LOWER_BOUND(_group, 1) TO UPPER_BOUND(_group, 1) DO
    (* Wieder prüfen, ob das aktuelle Element in der Gruppe ein gültiges Interface hat *)
    IF __QUERYINTERFACE(_group[_diFor1], _group[_diFor1]) THEN
        (* Überprüfen, ob das Mitglied für das Acknowledge relevant ist (d.h., ob es nicht ignoriert wird) *)
        IF NOT _group[_diFor1].IS_NOT_RELEVANT_TO_ACKNOWLEDGE THEN
            (* Wenn das Acknowledge des Mitglieds nicht dem erwarteten Zustand entspricht *)
            IF _group[_diFor1].acknowledge_substate <> _expectet_substate THEN
                (* Wenn der Zustand nicht dem erwarteten Zustand entspricht, setze den Gruppen-Check-Status auf den tatsächlichen Acknowledge-Wert des Mitglieds *)
                check_acknowledge_substate_of_group := _group[_diFor1].acknowledge_substate;
            END_IF;
        END_IF;
    END_IF;
END_FOR;
END_METHOD

ACTION RELEASE:
(* Set Release for each group and its components *)
FOR diFor1 := LOWER_BOUND(groups,1) TO UPPER_BOUND(groups,1) DO

    (* Check if group is in release state and not in lockdown *)
    IF (groups_en_release[diFor1] = en_release OR (groups_en_release[diFor1] = en_release_old AND (NOT xRelease OR groups_engine_acknowledged[diFor1] > 0 OR groups_engine_released[diFor1] > 0))) AND groups_en_acknowledge[diFor1] <> en_static_define_lockdown THEN
        (* Initially set group as ready for release *)
        AY_GROUPS_xReleaseCircuit[diFor1] := TRUE;
		groups_en_release[diFor1] := en_release;
		groups_en_release_substate[diFor1] 	:= en_release_substate;
        (* Check each member in the group to verify readiness for release *)
		IF __QUERYINTERFACE(groups[diFor1][0],TEMP_ITF_CIRCUIT) THEN
			IF TEMP_ITF_CIRCUIT.IS_RELEVANT_TO_RELEASE THEN		
				FOR diFor2 := LOWER_BOUND(groups[diFor1],1)+1 TO UPPER_BOUND(groups[diFor1],1) DO
					IF __QUERYINTERFACE(groups[diFor1][diFor2], TEMP_ITF_HYDRA) THEN
						IF NOT groups[diFor1][diFor2].IS_NOT_RELEVANT_TO_RELEASE AND NOT groups[diFor1][diFor2].IS_NOT_RELEVANT_TO_ACKNOWLEDGE THEN
							IF groups[diFor1][diFor2].acknowledge <> en_release OR groups[diFor1][diFor2].acknowledge_substate <> en_static_define_engine_release_from_substate THEN
								(* Member not ready, set group as not ready *)
								AY_GROUPS_xReleaseCircuit[diFor1] := FALSE;
							END_IF;
						END_IF;
					END_IF;
				END_FOR;
			END_IF;
		END_IF;
        (* Apply release settings to each relevant member of the group *)
        FOR diFor2 := LOWER_BOUND(groups[diFor1],1)+1 TO UPPER_BOUND(groups[diFor1],1) DO
            IF __QUERYINTERFACE(groups[diFor1][diFor2], groups[diFor1][diFor2]) THEN
                IF NOT groups[diFor1][diFor2].IS_NOT_RELEVANT_TO_RELEASE THEN
                    IF __QUERYINTERFACE(groups[diFor1][diFor2], TEMP_ITF_HYDRA) THEN
                        TEMP_ITF_HYDRA.set_release(en_release);
                        TEMP_ITF_HYDRA.set_release_substate(en_release_substate);
                        TEMP_ITF_HYDRA.set_release_next(en_release_next);
                    END_IF;
                ELSE
                    (* Member not relevant → set off *)
                    IF __QUERYINTERFACE(groups[diFor1][diFor2], TEMP_ITF_HYDRA) THEN
                        TEMP_ITF_HYDRA.set_release(en_static_define_state_off);
                        TEMP_ITF_HYDRA.set_release_substate(en_static_define_sub_state_off);
                        TEMP_ITF_HYDRA.set_release_next(en_release_next);
                    END_IF;
                END_IF;
            END_IF;
        END_FOR;

        (* Release settings for group leader *)
        IF groups[diFor1][LOWER_BOUND(groups[diFor1],1)] <> 0 THEN
            IF __QUERYINTERFACE(groups[diFor1][LOWER_BOUND(groups[diFor1],1)], TEMP_ITF_CIRCUIT) THEN
				TEMP_ITF_CIRCUIT.set_release(en_release);
				TEMP_ITF_CIRCUIT.set_release_substate(en_release_substate);
				TEMP_ITF_CIRCUIT.set_release_next(en_release_next);
			END_IF;
        END_IF;

    ELSE
        (* Group not in release → mark as not ready *)
        AY_GROUPS_xReleaseCircuit[diFor1] := FALSE;

        (* Turn off all members of the group *)
        FOR diFor2 := LOWER_BOUND(groups[diFor1],1) TO UPPER_BOUND(groups[diFor1],1) DO
            IF __QUERYINTERFACE(groups[diFor1][diFor2], TEMP_ITF_CIRCUIT) THEN
				TEMP_ITF_CIRCUIT.set_release(SEL(en_release = en_static_define_lockdown,en_static_define_state_off,en_static_define_lockdown));
				TEMP_ITF_CIRCUIT.set_release_substate(en_static_define_sub_state_off);
				TEMP_ITF_CIRCUIT.set_release_next(en_release_next);

            ELSIF __QUERYINTERFACE(groups[diFor1][diFor2], TEMP_ITF_HYDRA) THEN
                (* Check if member is part of any other released circuit before turning off *)
                lock_if_released_in_other_circuit := FALSE;
                FOR diFor3 := LOWER_BOUND(groups,1) TO UPPER_BOUND(groups,1) DO
                    IF TEMP_ITF_HYDRA.MEMBER_OF(TO_USINT(diFor3)) AND (groups_en_release[diFor3] = en_release OR groups_en_release[diFor3] = en_release_old) AND groups_en_acknowledge[diFor3] <> en_static_define_lockdown THEN
                        lock_if_released_in_other_circuit := TRUE;
                    END_IF;
                END_FOR;
                IF NOT lock_if_released_in_other_circuit THEN
					TEMP_ITF_HYDRA.set_release(SEL(en_release = en_static_define_lockdown,en_static_define_state_off,en_static_define_lockdown));
					TEMP_ITF_HYDRA.set_release_substate(en_static_define_sub_state_off);
					TEMP_ITF_HYDRA.set_release_next(en_release_next);
                END_IF;
            END_IF;
        END_FOR;
    END_IF;
END_FOR;
END_ACTION

// Methode zum Setzen des Release-Status für alle relevanten Elemente einer Gruppe
METHOD set_release_of_group

VAR_INPUT
    // Array dynamischer Größe mit Objekten, die das Interface ITF_GROUPBASE implementieren
    _group : ARRAY[*] OF ITF_GROUPBASE;
    
    // Neuer Release-Zustand, der für alle relevanten Gruppenobjekte gesetzt werden soll
    _state : INT;
END_VAR

VAR
    // Laufvariable für die Schleifeniteration über _group
    _diFor1 : DINT;
END_VAR
// Durchlaufe alle Elemente der ersten Dimension von _group
FOR _diFor1 := LOWER_BOUND(_group, 1) TO UPPER_BOUND(_group, 1) DO

    // Prüft, ob das aktuelle Element das erwartete Interface implementiert
    IF __QUERYINTERFACE(_group[_diFor1], _group[_diFor1]) THEN

        // Verarbeitung nur durchführen, wenn das Element für den Release-Prozess relevant ist
        IF NOT _group[_diFor1].IS_NOT_RELEVANT_TO_RELEASE THEN
            
            // Setzt den Release-Status des Elements entsprechend dem übergebenen Zustand
            _group[_diFor1].set_release(_state);
        END_IF;
    END_IF;
END_FOR;
END_METHOD

// Methode zum Setzen eines Sub-Release-Status für alle relevanten Elemente einer Gruppe
METHOD set_release_substate_of_group

VAR_INPUT
    // Array variabler Größe mit Objekten, die das Interface ITF_GROUPBASE implementieren
    _group : ARRAY[*] OF ITF_GROUPBASE;
    
    // Sub-Release-Zustand, der für alle relevanten Gruppenobjekte gesetzt werden soll
    _sub_state : INT;
END_VAR

VAR
    // Laufvariable für die Iteration über das Gruppen-Array
    _diFor1 : DINT;
END_VAR
// Durchlaufe alle Elemente der ersten Dimension von _group
FOR _diFor1 := LOWER_BOUND(_group, 1) TO UPPER_BOUND(_group, 1) DO

    // Prüft, ob das aktuelle Element das erwartete Interface implementiert
    IF __QUERYINTERFACE(_group[_diFor1], _group[_diFor1]) THEN

        // Verarbeitung nur durchführen, wenn das Element für den Release-Prozess relevant ist
        IF NOT _group[_diFor1].IS_NOT_RELEVANT_TO_RELEASE THEN
            
            // Setzt den Release-Status des Elements entsprechend dem übergebenen Zustand
            _group[_diFor1].set_release_substate(_sub_state);
		ELSE
	        // Setzt den Release-Status des Elements entsprechend dem übergebenen Zustand
            _group[_diFor1].set_release_substate(en_static_define_sub_state_off);	 	
        END_IF;
    END_IF;
END_FOR;
END_METHOD

// Methode zum Setzen des Release-Status für alle relevanten Elemente einer Gruppe
METHOD set_release_next_of_group

VAR_INPUT
    // Array dynamischer Größe mit Objekten, die das Interface ITF_GROUPBASE implementieren
    _group : ARRAY[*] OF ITF_GROUPBASE;
    
    // Neuer Release-Zustand, der für alle relevanten Gruppenobjekte gesetzt werden soll
    _state : INT;
END_VAR

VAR
    // Laufvariable für die Schleifeniteration über _group
    _diFor1 : DINT;
END_VAR
// Durchlaufe alle Elemente der ersten Dimension von _group
FOR _diFor1 := LOWER_BOUND(_group, 1) TO UPPER_BOUND(_group, 1) DO

    // Prüft, ob das aktuelle Element das erwartete Interface implementiert
    IF __QUERYINTERFACE(_group[_diFor1], _group[_diFor1]) THEN
  
		// Setzt den Release-Status des Elements entsprechend dem übergebenen Zustand
		_group[_diFor1].set_release_next(_state);
    END_IF;
END_FOR;
END_METHOD

ACTION LOCKDOWN:
(* Get Status LockDown Engine*)
uiCountEngineLockDown := 0;
FOR diFor1 := LOWER_BOUND(groups,1) TO UPPER_BOUND(groups,1) DO
	IF __QUERYINTERFACE(groups[diFor1][LOWER_BOUND(groups[diFor1],1)],TEMP_ITF_CIRCUIT) THEN
		uiCountEngineLockDown := uiCountEngineLockDown + TEMP_ITF_CIRCUIT.GET_ANZ_LOCKDOWN;
	END_IF;
END_FOR;
END_ACTION

ACTION AVAIABLE:
IF en_check = en_check_old AND en_check_substate = en_check_substate_old THEN
    iAvailableTemp := 0;

    FOR diFor1 := LOWER_BOUND(groups, 1) TO UPPER_BOUND(groups, 1) DO
        // Gruppenstatus prüfen
        groups_en_available[diFor1] := check_available_of_group(diFor1, groups[diFor1], en_check);
        groups_en_available_substate[diFor1] := check_available_substate_of_group(diFor1, groups[diFor1], en_check_substate);

        // Anzahl verfügbarer Engines ermitteln
        IF __QUERYINTERFACE(groups[diFor1][LOWER_BOUND(groups[diFor1],1)], TEMP_ITF_CIRCUIT) THEN
            groups_engine_available[diFor1] := TO_INT(TEMP_ITF_CIRCUIT.GET_ANZ_AVAIABLE);
        ELSE
            groups_engine_available[diFor1] := 0;
        END_IF;

        // Summierung verfügbarer Engines
        iAvailableTemp := iAvailableTemp + groups_engine_available[diFor1];
    END_FOR;
	iAvailable := iAvailableTemp;
	
	FOR diFor1 := LOWER_BOUND(groups, 1) TO UPPER_BOUND(groups, 1) DO
        // Aggregation des Managerstatus
        IF groups_en_available[diFor1] = en_check AND groups_en_available_substate[diFor1] = en_check_substate THEN
            en_available := en_check;
            en_available_substate := en_check_substate;
			RETURN;
		END_IF
	END_FOR;
	FOR diFor1 := LOWER_BOUND(groups, 1) TO UPPER_BOUND(groups, 1) DO
    	IF groups_en_available[diFor1] = en_static_define_state_not_ready AND groups_en_available_substate[diFor1] = en_check_substate THEN
            en_available := en_static_define_state_not_ready;
            en_available_substate := en_check_substate;
			RETURN;
		END_IF;
	END_FOR;	
	FOR diFor1 := LOWER_BOUND(groups, 1) TO UPPER_BOUND(groups, 1) DO
		IF  groups_en_available[diFor1] <> en_static_define_lockdown AND groups_en_available_substate[diFor1] = en_check_substate THEN
		    en_available := groups_en_available[diFor1];
            en_available_substate := en_check_substate;	
			RETURN;
		END_IF;
	END_FOR;
	en_available := en_static_define_lockdown;
	en_available_substate := en_check_substate;	
END_IF;
END_ACTION

(* Methode, die den avaiable-Zustand aller Mitglieder einer Gruppe überprüft und den Status der Gruppe zurückgibt *)
METHOD check_available_of_group : INT
VAR_INPUT
	_group_nr			 : DINT;	// Gruppennummer als Info
    (* Eingabeparameter: Eine Array von Gruppenmitgliedern (Interface vom Typ ITF_GROUPBASE) *)
    _group               : ARRAY[*] OF ITF_GROUPBASE;
    
    (* Eingabeparameter: Der erwartete avaiable-Zustand, auf den alle Mitglieder überprüft werden *)
    _expectet_state      : INT;
END_VAR

VAR
    (* Interne Variable für die Schleifenindizierung *)
    _diFor1              : DINT;
END_VAR
(* Initialisierung des Check-Status der Gruppe auf "lockdown" *)
check_available_of_group := en_static_define_lockdown;

(* Iteration durch alle Mitglieder der Gruppe, um zu überprüfen ob Mitglider vorhanden*)
FOR _diFor1 := LOWER_BOUND(_group, 1) TO UPPER_BOUND(_group, 1) DO
    (* Prüfen, ob das aktuelle Element in der Gruppe ein gültiges Interface hat *)
    IF __QUERYINTERFACE(_group[_diFor1], _group[_diFor1]) THEN
        (* Wenn das Interface gültig ist, setze den Check-Status nicht bereit *)
        check_available_of_group := en_static_define_state_not_ready;
    END_IF;
END_FOR;

(* Iteration durch alle Mitglieder der Gruppe, um den erwarteten Zustand zu überprüfen *)
FOR _diFor1 := LOWER_BOUND(_group, 1) TO UPPER_BOUND(_group, 1) DO
    (* Prüfen, ob das aktuelle Element in der Gruppe ein gültiges Interface hat *)
    IF __QUERYINTERFACE(_group[_diFor1], _group[_diFor1]) THEN
        (* Wenn das Interface gültig ist, setze den Check-Status auf den erwarteten Zustand *)
        check_available_of_group := _expectet_state;
    END_IF;
END_FOR;

(* Iteration durch alle Mitglieder der Gruppe, um den Zustand jedes Mitglieds zu überprüfen und den Gruppenstatus anzupassen *)
FOR _diFor1 := LOWER_BOUND(_group, 1) TO UPPER_BOUND(_group, 1) DO
    (* Wieder prüfen, ob das aktuelle Element in der Gruppe ein gültiges Interface hat *)
    IF __QUERYINTERFACE(_group[_diFor1], _group[_diFor1]) THEN
        (* Überprüfen, ob das Mitglied für das avaiable relevant ist (d.h., ob es nicht ignoriert wird) *)
        IF NOT _group[_diFor1].IS_NOT_RELEVANT_TO_CHECK THEN
            (* Wenn das Acknowledge des Mitglieds nicht dem erwarteten Zustand entspricht *)
            IF _group[_diFor1].available <> _expectet_state THEN
                (* Wenn der Zustand nicht dem erwarteten Zustand entspricht, setze den Gruppen-Check-Status auf den tatsächlichen avaiable-Wert des Mitglieds *)
                check_available_of_group := _group[_diFor1].available;
                IF check_available_of_group = en_static_define_lockdown THEN
					EXIT;
				END_IF;
			END_IF;
        END_IF;
    END_IF;
END_FOR;
END_METHOD

(* Methode, die den avaiable-Zustand aller Mitglieder einer Gruppe überprüft und den Status der Gruppe zurückgibt *)
METHOD check_available_substate_of_group : INT
VAR_INPUT
	_group_nr			 : DINT;	// Gruppennummer als Info
    (* Eingabeparameter: Eine Array von Gruppenmitgliedern (Interface vom Typ ITF_GROUPBASE) *)
    _group               : ARRAY[*] OF ITF_GROUPBASE;
    
    (* Eingabeparameter: Der erwartete avaiable-Zustand, auf den alle Mitglieder überprüft werden *)
    _expectet_substate   : INT;
END_VAR

VAR
    (* Interne Variable für die Schleifenindizierung *)
    _diFor1              : DINT;
END_VAR
(* Initialisierung des Check-Status der Gruppe auf "Lockdown" *)
check_available_substate_of_group := en_static_define_sub_state_off;

(* Iteration durch alle Mitglieder der Gruppe, um den erwarteten Zustand zu überprüfen *)
FOR _diFor1 := LOWER_BOUND(_group, 1) TO UPPER_BOUND(_group, 1) DO
    (* Prüfen, ob das aktuelle Element in der Gruppe ein gültiges Interface hat *)
    IF __QUERYINTERFACE(_group[_diFor1], _group[_diFor1]) THEN
        (* Wenn das Interface gültig ist, setze den Check-Status auf den erwarteten Zustand *)
        check_available_substate_of_group := _expectet_substate;
    END_IF;
END_FOR;

(* Iteration durch alle Mitglieder der Gruppe, um den Zustand jedes Mitglieds zu überprüfen und den Gruppenstatus anzupassen *)
FOR _diFor1 := LOWER_BOUND(_group, 1) TO UPPER_BOUND(_group, 1) DO
    (* Wieder prüfen, ob das aktuelle Element in der Gruppe ein gültiges Interface hat *)
    IF __QUERYINTERFACE(_group[_diFor1], _group[_diFor1]) THEN
        (* Überprüfen, ob das Mitglied für das Acknowledge relevant ist (d.h., ob es nicht ignoriert wird) *)
        IF NOT _group[_diFor1].IS_NOT_RELEVANT_TO_CHECK THEN
            (* Wenn das Acknowledge des Mitglieds nicht dem erwarteten Zustand entspricht *)
            IF _group[_diFor1].available_substate <> _expectet_substate THEN
                (* Wenn der Zustand nicht dem erwarteten Zustand entspricht, setze den Gruppen-Check-Status auf den tatsächlichen avaiable-Wert des Mitglieds *)
                check_available_substate_of_group := _group[_diFor1].available_substate;
            END_IF;
        END_IF;
    END_IF;
END_FOR;
END_METHOD

METHOD ADD_CLIENT : BOOL
VAR_INPUT
	ITF_GROUP_BASE_IN	:	ITF_GROUPBASE;
END_VAR
VAR
	ITF_CIRCUIT_QUERRY	:	ITF_CIRCUIT;
	usiCircuitNr		:	USINT;
	ITF_HYDRA_QUERRY	:	ITF_HYDRA;
	xFailToAdd			:	BOOL;
	xExist				:	BOOL;
	xRegroup			:	BOOL;
	diForTemp1			:	DINT;
	diForTemp2			:	DINT;
	diForTemp3			:	DINT;
	diAddIn				:	DINT;
END_VAR
(* ADD CIRCUIT *)
IF __QUERYINTERFACE(ITF_GROUP_BASE_IN,ITF_CIRCUIT_QUERRY) THEN
	usiCircuitNr := ITF_CIRCUIT_QUERRY.CIRCUIT_NR;
	IF usiCircuitNr >= 1 AND usiCircuitNr <= GVL_CONSTANT.MAX_GROUPS THEN 
		IF groups[usiCircuitNr][0] = 0 THEN
			__QUERYINTERFACE(ITF_CIRCUIT_QUERRY,groups[usiCircuitNr][0]);
			ITF_CIRCUIT_QUERRY.IS_ADDED_TO_NESSESARY := TRUE;
		ELSIF groups[usiCircuitNr][0] = ITF_GROUP_BASE_IN THEN
			ADD_CLIENT := TRUE;	
			ITF_CIRCUIT_QUERRY.IS_ADDED_TO_NESSESARY := TRUE;
		ELSE
			ADD_CLIENT := FALSE;
			ITF_CIRCUIT_QUERRY.IS_ADDED_TO_NESSESARY := FALSE;
		END_IF;
	END_IF;
(* ADD HYDRA *)
ELSIF __QUERYINTERFACE(ITF_GROUP_BASE_IN,ITF_HYDRA_QUERRY) THEN
	(* Check if is ADDED *)
	IF NOT ITF_HYDRA_QUERRY.IS_ADDED_TO_NESSESARY THEN
		FOR diForTemp1 := LOWER_BOUND(groups,1) TO UPPER_BOUND(groups,1) DO
			(* Reset Exist *)
			xExist := FALSE;
			(* Get Group Member *)
			IF ITF_HYDRA_QUERRY.MEMBER_OF(TO_USINT(diForTemp1)) THEN
				FOR diForTemp2 := LOWER_BOUND(groups[diForTemp1],1) TO UPPER_BOUND(groups[diForTemp1],1) DO
					IF groups[diForTemp1][diForTemp2] = ITF_GROUP_BASE_IN THEN
						xExist  := TRUE;
					END_IF;
				END_FOR;
				(* Add if not Exist *)
				IF NOT xExist THEN 
					IF sync_groups[diForTemp1] <> 0 THEN
						diAddIn  := __XADD(ADR(sync_groups[diForTemp1]),1);
						IF diAddIn >= 1 AND diAddIn <= UPPER_BOUND(groups[diForTemp1],1) THEN
							__QUERYINTERFACE(ITF_HYDRA_QUERRY,groups[diForTemp1][diAddIn]);
						ELSE
							xFailToAdd := TRUE;	
							ADD_CLIENT := FALSE;
						END_IF
					ELSE	
						xFailToAdd := TRUE;
						ADD_CLIENT := FALSE;
					END_IF;
				END_IF;
			ELSE
				FOR diForTemp2 := LOWER_BOUND(groups[diForTemp1],1) TO UPPER_BOUND(groups[diForTemp1],1) DO
					IF groups[diForTemp1][diForTemp2] = ITF_GROUP_BASE_IN THEN
						groups[diForTemp1][diForTemp2] := 0;
						FOR diForTemp3 := diForTemp2 TO UPPER_BOUND(groups[diForTemp1],1)-1 DO 
							groups[diForTemp1][diForTemp3] := groups[diForTemp1][diForTemp3+1];	
						END_FOR
						diAddIn  := __XADD(ADR(sync_groups[diForTemp1]),-1);
					END_IF;
				END_FOR;				
			END_IF
		END_FOR;
		ITF_HYDRA_QUERRY.IS_ADDED_TO_NESSESARY := NOT xFailToAdd;
	END_IF;	
ELSE
	ADD_CLIENT := FALSE;
END_IF;
END_METHOD

ACTION actParameter:
fbConfigFile();

scParameter.fbiTypeOfEngineManagement	(_usiParaNr := 1,	_WertInit := 0,		_MinInit := 0,	_MaxInit := 2,	itfConfigFb := fbConfigFile);
scParameter.fbtZuschaltSperrzeit		(_usiParaNr := 2,	_WertInit := T#5M,	_MinInit :=  ,	_MaxInit :=	 ,	itfConfigFb := fbConfigFile);
END_ACTION

//FB_Init ist immer implizit verfügbar und wird primär für die Initialisierung verwendet.
//Der Rückgabewert wird nicht ausgewertet. Für gezielte Einflussnahme können Sie
//die Methoden explizit deklarieren und darin mit dem Standard-Initialisierungscode 
//zusätzlichen Code bereitstellen. Sie können den Rückgabewert auswerten.
METHOD FB_Init: BOOL
VAR_INPUT    
bInitRetains: BOOL; // TRUE: Die Retain-Variablen werden initialisiert (Reset warm / Reset kalt)    
bInCopyCode: BOOL;  // TRUE: Die Instanz wird danach in den Kopiercode kopiert (Online-Change)
END_VAR
END_METHOD

ACTION DEMAND:
(* Get Demand of Group *)
FOR diFor1 := LOWER_BOUND(groups,1) TO UPPER_BOUND(groups,1) DO
	// setze auf ignore
	groups_en_demand[diFor1] := en_static_define_state_ignore;
	// Iteriere grouppen
	FOR diFor2 := LOWER_BOUND(groups[diFor1],1) TO UPPER_BOUND(groups[diFor1],1) DO
		// Prüfe Interface
		IF __QUERYINTERFACE(groups[diFor1][diFor2],TEMP_ITF_GROUPBASE) THEN
			// setze erstes demand
			IF groups_en_demand[diFor1] = en_static_define_state_ignore THEN
				groups_en_demand[diFor1] := TEMP_ITF_GROUPBASE.demand;
			ELSE
				// Prüfe auf höher priorisiertes demand
				FOR diFor3 := LOWER_BOUND(priority_array,1) TO UPPER_BOUND(priority_array,1) DO
					IF groups_en_demand[diFor1] = priority_array[diFor3] THEN
						EXIT;
					ELSIF TEMP_ITF_GROUPBASE.demand = priority_array[diFor3] THEN
						groups_en_demand[diFor1] := TEMP_ITF_GROUPBASE.demand;
						EXIT;
					END_IF
				END_FOR;			
			END_IF;
		END_IF;	
	END_FOR;
END_FOR;

(* Get Demand on all groups *)
en_demand := en_static_define_state_ignore;
FOR diFor1 := LOWER_BOUND(groups_en_demand,1) TO UPPER_BOUND(groups_en_demand,1) DO
	// setze erstes demand
	IF en_demand = en_static_define_state_ignore THEN
		en_demand := groups_en_demand[diFor1];
	ELSE
		// Prüfe auf höher priorisiertes demand
		FOR diFor3 := LOWER_BOUND(priority_array,1) TO UPPER_BOUND(priority_array,1) DO
			IF en_demand = priority_array[diFor3] THEN
				EXIT;
			ELSIF groups_en_demand[diFor1] = priority_array[diFor3] THEN
				en_demand := groups_en_demand[diFor1];
				EXIT;
			END_IF
		END_FOR;			
	END_IF;
END_FOR;
END_ACTION

METHOD set_priority_array
VAR_INPUT
	priority	:	INT;
	state		:	INT;
END_VAR
IF TO_DINT(priority) >= LOWER_BOUND(priority_array,1) AND TO_DINT(priority) <= UPPER_BOUND(priority_array,1) THEN
	priority_array[priority] := state;
END_IF;
END_METHOD

METHOD init_priority_array_with_ignore_state
VAR_INPUT
	ignore_state		:	INT;
END_VAR
VAR
	_diFor1 :	DINT;
END_VAR
FOR _diFor1 := LOWER_BOUND(priority_array,1) TO UPPER_BOUND(priority_array,1) DO
	priority_array[_diFor1] := ignore_state;
END_FOR;
END_METHOD

END_FUNCTION_BLOCK

